Yaskawa INFORM job: X2_34-37(-90,0)_HARDOX.JBI

/JOB
//NAME X2_34-37(-90,0)_HARDOX
//POS
///NPOS 543,543,543,15,0,0
///TOOL 0
///POSTYPE PULSE
///PULSE
C00000=-109615,-71844,-36862,18422,13388,2271
C00001=-107008,40287,15446,7646,74688,11911
C00002=-107149,45804,24218,7788,72161,11701
C00003=-108392,48192,28010,10243,72680,1076
C00004=-108392,48392,29954,10302,71604,983
C00005=-108392,48331,29423,10286,71896,1009
C00006=-108010,50265,31522,10186,71551,1114
C00007=-108392,48331,29423,10286,71896,1009
C00008=-108911,49901,30550,10443,72076,8021
C00009=-109414,51873,32709,10619,71831,7821
C00010=-108911,49901,30550,10443,72076,8021
C00011=-102203,43615,23227,8248,72569,10434
C00012=-106081,49085,29485,15378,74997,2308
C00013=-106081,49206,30588,15419,74401,2232
C00014=-106081,49153,30130,15402,74647,2263
C00015=-105730,50968,32108,15326,74307,2347
C00016=-106081,49153,30130,15402,74647,2263
C00017=-108167,43461,21271,12324,74506,6920
C00018=-107374,42085,15448,7738,75637,11845
C00019=-120191,30165,1303,6226,81332,-6626
C00020=-119709,34887,8992,6124,79003,-6581
C00021=-119523,36874,12198,6088,78043,-6565
C00022=-119519,36825,13807,6108,77033,-6613
C00023=-119523,36874,12198,6088,78043,-6565
C00024=-119515,36764,13496,6103,77191,-6604
C00025=-119868,39633,16467,6214,76866,-6741
C00026=-119515,36764,13496,6103,77191,-6604
C00027=-121889,32841,7793,6759,78864,-7323
C00028=-122776,40716,17165,7052,77228,-7717
C00029=-121823,41691,18182,6780,77023,-7402
C00030=-122776,40716,17165,7052,77228,-7717
C00031=-121889,32783,9008,6775,78090,-7366
C00032=-119523,36874,12198,6088,78043,-6565
C00033=-119709,34887,8992,6124,79003,-6581
C00034=-120191,30165,1303,6226,81332,-6626
C00035=-121604,30205,1144,6630,81559,-7083
C00036=-121089,34887,8794,6520,79231,-7034
C00037=-120696,52216,26132,6337,84983,-6608
C00038=-120696,52210,26931,6339,84491,-6634
C00039=-120890,37827,12979,6483,78156,-7023
C00040=-120878,38017,14560,6499,77285,-7064
C00041=-121214,39658,16269,6601,77105,-7189
C00042=-120878,38555,15116,6500,77220,-7067
C00043=-120100,37082,13567,6272,77355,-6796
C00044=-119528,38122,14634,6107,77190,-6608
C00045=-120486,37092,12834,6373,77838,-6903
C00046=-120682,35058,10322,6419,78351,-6942
C00047=-121186,30266,2562,6523,80690,-6990
C00048=-134026,40869,15057,-4047,52311,-47824
C00049=-133273,45805,23219,-4742,49872,-47398
C00050=-131154,47390,26558,-10411,48349,-46747
C00051=-131420,50658,30105,-10292,47819,-46809
C00052=-130698,69773,43023,-10534,62516,-48132
C00053=-130716,70192,44349,-10580,61922,-48084
C00054=-130716,70230,44981,-10614,61557,-48050
C00055=-130716,70169,43891,-10554,62186,-48109
C00056=-134669,50089,27300,-4593,51640,-48236
C00057=-135826,53842,33106,-2979,47876,-48446
C00058=-135153,55159,34569,-3502,47681,-48138
C00059=-135859,54027,33595,-2932,47595,-48448
C00060=-135721,50610,29531,-3003,48343,-48409
C00061=-134026,40869,15057,-4047,52311,-47824
C00062=-158164,35728,9631,12841,54320,-57618
C00063=-156933,39530,16487,12369,51918,-57402
C00064=-155249,48901,23783,8538,56742,-56466
C00065=-155249,48910,25069,8614,55964,-56530
C00066=-156452,41160,19364,12190,50934,-57317
C00067=-155375,36976,18106,9951,45044,-57856
C00068=-155421,38663,19846,10021,44849,-57900
C00069=-156479,41060,19769,12260,50644,-57365
C00070=-160744,48197,26791,24242,55405,-57248
C00071=-159861,48269,26866,23741,55141,-56924
C00072=-161011,41761,19928,24147,56321,-57142
C00073=-157483,35375,10637,12509,53434,-57446
C00074=-160593,39475,13550,14508,54241,-58615
C00075=-159342,43270,20469,14089,51785,-58436
C00076=-157654,61041,34307,9103,61397,-56807
C00077=-157654,61062,35619,9172,60610,-56871
C00078=-157654,61044,34661,9122,61183,-56824
C00079=-156017,38846,20879,6547,42814,-58158
C00080=-156075,40278,22364,6619,42641,-58197
C00081=-156484,37577,19565,6938,43009,-58369
C00082=-158359,40577,22676,8640,42818,-59307
C00083=-163736,54420,35453,24006,50522,-59362
C00084=-163085,54943,36034,23619,50253,-59126
C00085=-163861,53390,33193,23805,51349,-59211
C00086=-160593,39475,13550,14508,54241,-58615
C00087=-148971,42504,16746,4915,52183,-53021
C00088=-147979,47046,24523,4355,49683,-52716
C00089=-147593,48996,27807,4132,48646,-52593
C00090=-147590,49137,29621,4197,47605,-52637
C00091=-147593,48996,27807,4132,48646,-52593
C00092=-147610,49163,29309,4198,47810,-52637
C00093=-147661,52475,32942,4273,47281,-52683
C00094=-147610,49163,29309,4198,47810,-52637
C00095=-147454,49128,29272,4080,47808,-52567
C00096=-147457,49325,29466,4083,47790,-52569
C00097=-146486,49526,29681,3347,47716,-52137
C00098=-147457,49325,29466,4083,47790,-52569
C00099=-147454,49128,29272,4080,47808,-52567
C00100=-147593,48996,27807,4132,48646,-52593
C00101=-147979,47046,24523,4355,49683,-52716
C00102=-148753,37651,9035,4624,54413,-52827
C00103=-143332,14237,-19618,-15194,67693,-56285
C00104=-143234,13815,-14606,-15619,64520,-55819
C00105=-143234,13420,-12421,-15818,63029,-55609
C00106=-143234,13266,-11275,-15925,62274,-55501
C00107=-143234,13282,-11406,-15913,62359,-55513
C00108=-142905,14636,-10175,-16100,62361,-55388
C00109=-143057,13626,-13166,-15840,63606,-55626
C00110=-122407,-4916,-29077,-25933,68954,-48837
C00111=-79716,14771,-17940,-28940,82202,-34377
C00112=-81521,13206,-15483,-28515,79567,-34389
C00113=-81521,12956,-14255,-28586,78787,-34193
C00114=-81536,13061,-14375,-28568,78899,-34239
C00115=-81552,13376,-14091,-28564,78881,-34239
C00116=-81324,12822,-15528,-28589,79487,-34301
C00117=-153828,-54456,-66092,3136,64230,-58148
C00118=-168903,-101217,-87597,11823,54897,-64642
C00119=-187075,-120078,-80481,24912,5471,-74731
C00120=-125084,-120078,-92282,24912,5045,-74731
C00121=-122155,56416,27906,-88,21317,-63492
C00122=-122155,75596,27906,-2527,72055,-63492
C00123=-129231,63588,14742,9851,74193,-63747
C00124=-129934,64141,19195,10317,71853,-64173
C00125=-129934,63674,20017,10359,71118,-64236
C00126=-129934,63737,19901,10353,71221,-64227
C00127=-129659,64892,21241,10232,70961,-64158
C00128=-129934,64415,18756,10296,72257,-64138
C00129=-132222,69706,24963,11475,71461,-64978
C00130=-132222,69058,26180,11545,70402,-65080
C00131=-131900,68421,25429,11378,70491,-64961
C00132=-131996,66718,21836,11340,71814,-64867
C00133=-130068,63875,18521,10367,72141,-64191
C00134=-129934,63737,19901,10353,71221,-64227
C00135=-129659,64892,21241,10232,70961,-64158
C00136=-129936,63793,17790,10283,72529,-64117
C00137=-88784,58262,10938,-10282,73900,-50815
C00138=-84208,56991,12900,-3171,67181,-46725
C00139=-84435,57608,15935,-3079,65626,-46760
C00140=-84435,57210,16828,-3097,64873,-46739
C00141=-84435,57270,16685,-3094,64991,-46743
C00142=-84516,58633,18225,-3054,64742,-46763
C00143=-84215,57626,14285,-3179,66658,-46710
C00144=-88784,58262,10938,-10282,73900,-50815
C00145=-130230,57807,7300,10270,75892,-63928
C00146=-119131,59701,11284,-18823,72688,-66064
C00147=-121021,64874,21663,-18257,68751,-66091
C00148=-121021,64408,22622,-18356,67963,-65965
C00149=-121021,64908,21591,-18251,68811,-66098
C00150=-119131,67163,24223,-19268,68781,-65421
C00151=-119066,66124,24431,-19384,68169,-65294
C00152=-119315,66407,24761,-19266,68060,-65365
C00153=-119315,66969,23588,-19142,69017,-65526
C00154=-121021,64979,21457,-18238,68923,-66116
C00155=-121021,64479,22465,-18340,68089,-65984
C00156=-120883,66044,24287,-18448,67818,-65890
C00157=-120883,66039,23301,-18376,68392,-65982
C00158=-125359,68164,24258,-15996,67985,-67508
C00159=-125355,67935,25342,-16085,67231,-67400
C00160=-125355,67510,26289,-16176,66462,-67291
C00161=-125355,67568,26150,-16162,66575,-67307
C00162=-125232,69006,27841,-16263,66308,-67224
C00163=-125264,67856,24082,-16054,67958,-67468
C00164=-118603,65727,21589,-19430,69736,-65391
C00165=-117191,86264,44946,-23194,75505,-66935
C00166=-117189,86115,44761,-23192,75540,-66941
C00167=-117189,86115,44761,-23192,75540,-66941
C00168=-117506,84477,42726,-23036,75832,-67112
C00169=-117132,73456,32688,-25561,71261,-66383
C00170=-118175,73897,33217,-25111,70866,-66682
C00171=-123739,77574,37647,-22686,68558,-68266
C00172=-123019,74931,32102,-22743,70649,-68420
C00173=-118383,77560,28081,-24424,75407,-67742
C00174=-128287,78191,30299,3222,75938,-66053
C00175=-128503,77276,32915,3346,73869,-66179
C00176=-128483,76731,32333,3336,73949,-66169
C00177=-128483,76731,32333,3336,73949,-66169
C00178=-128335,75085,30341,3266,74321,-66111
C00179=-127967,73943,28963,3095,74566,-65984
C00180=-126238,72254,26940,2321,74892,-65413
C00181=-107561,64945,18412,-6002,76780,-59423
C00182=-95850,66897,26093,8333,67040,-51862
C00183=-95804,66521,24248,8255,67969,-51781
C00184=-109126,32483,-12900,14644,74981,-55562
C00185=-109126,32483,-12900,14644,28895,-55562
C00186=-105965,-15733,-41727,12755,21555,-55066
C00187=-95466,-93835,-85705,-21780,8598,-39995
C00188=-117456,-93835,-85705,-3320,8456,-83429
C00189=-140967,-12970,-52901,4588,62048,-69725
C00190=-151426,22553,-30287,8605,79970,-63791
C00191=-170197,65047,13937,16074,97750,-54995
C00192=-169007,70240,20067,15770,96475,-54777
C00193=-175404,86334,34832,19373,106938,-55773
C00194=-174173,83341,34513,19133,105400,-55601
C00195=-179433,56900,11422,30057,94253,-55502
C00196=-178535,49502,4014,27996,88823,-56876
C00197=-179527,69319,26237,30671,91177,-56324
C00198=-179117,69620,25739,29739,90864,-56355
C00199=-180097,67994,26330,32410,86483,-57198
C00200=-174100,64042,14056,17976,91926,-56289
C00201=-175447,65123,11808,18399,94042,-56406
C00202=-164161,72,-39985,-6764,90046,-34295
C00203=-130432,-55243,-47386,-13424,82603,8412
C00204=-110572,-56965,-55890,-14658,90278,14468
C00205=-134387,-39172,-38807,12376,86277,-20344
C00206=-136266,-41846,-34601,16059,78566,-27361
C00207=-135424,-39022,-31748,15965,78109,-27121
C00208=-132144,-43884,-34748,15569,76844,-26110
C00209=-133349,-52476,-37829,19150,70304,-22714
C00210=-132707,-53219,-38228,19044,70026,-22517
C00211=-133874,-49344,-36092,21066,73724,-26553
C00212=-127403,-56601,-39797,20204,70737,-24655
C00213=-130575,-58808,-42172,20683,71834,-25657
C00214=-131419,-52897,-41760,13173,72105,-2236
C00215=-151757,-37235,-32664,25855,92713,-16023
C00216=-148694,-31120,-30848,28555,97484,-16481
C00217=-152363,20888,-11521,23566,108052,-25705
C00218=-155491,63274,13853,18429,111086,-34801
C00219=-150514,89045,46229,21307,107758,-32982
C00220=-149106,88504,48693,21100,105732,-32842
C00221=-152517,63826,23946,30540,100235,-10367
C00222=-144965,57793,12440,13988,97767,-10863
C00223=-145698,58452,15092,12206,89625,-12161
C00224=-143897,56959,13401,8510,88242,-7863
C00225=-138738,54288,10428,-948,87223,2685
C00226=-138154,54736,10996,-4550,87493,6522
C00227=-140559,38499,-1659,880,75847,28463
C00228=-140619,46287,2526,1728,82676,28626
C00229=-139837,43342,-3801,1439,85041,28899
C00230=-141798,27002,-27786,2149,91441,28405
C00231=-143772,-19107,-38740,14355,94017,-12677
C00232=-143698,-35148,-33847,20276,92427,-33189
C00233=-141918,-24797,-26817,20326,92921,-32464
C00234=-139594,-23350,-22642,20301,90627,-32011
C00235=-137429,-46971,-35033,19650,72370,-30958
C00236=-130857,-51491,-37639,10003,64087,-16893
C00237=-124996,-53139,-38566,2264,61948,-7877
C00238=-114020,-50430,-37038,-13344,65966,10499
C00239=-112071,-46775,-34852,-17581,69897,16673
C00240=-117935,-60108,-42034,-7672,56240,37337
C00241=-115664,-65010,-47736,-8512,57449,38158
C00242=-121785,-61828,-52329,-5505,69210,35118
C00243=-148930,-33628,-41038,4538,77484,18447
C00244=-163858,24222,1645,10794,81228,7547
C00245=-163712,28964,9442,10824,78886,7392
C00246=-163731,31317,12909,10857,77980,7305
C00247=-164778,31926,13518,11115,78061,6949
C00248=-169796,40183,22289,16135,80950,-18095
C00249=-170946,41436,24303,16621,77711,-36979
C00250=-169129,60932,43860,12206,77205,-36613
C00251=-174700,53660,39403,25265,70725,-61619
C00252=-176244,52382,34806,25393,73168,-61673
C00253=-174832,57379,31343,14926,87681,-59388
C00254=-147451,1111,-29714,5377,100632,-19781
C00255=-112791,-31989,-50015,-2241,90212,24459
C00256=-107981,-35875,-46971,-4517,78040,26268
C00257=-109410,-31915,-41181,-4141,76439,25836
C00258=-109671,-29943,-38250,-4081,75635,25773
C00259=-108634,-25346,-36028,-8315,81190,19632
C00260=-113738,-28838,-38579,-3049,79626,8435
C00261=-120146,-28716,-38356,4151,79685,-1679
C00262=-130395,-15154,-28625,15552,87688,-20481
C00263=-128753,-14804,-28536,10287,83416,-20949
C00264=-132110,-20936,-30028,13610,74111,-31363
C00265=-127631,-24253,-35023,5775,74490,-30240
C00266=-129181,-27934,-40726,6212,76213,-30690
C00267=-139651,-3107,-33687,4364,86662,15844
C00268=-140099,618,-27389,4493,84729,15631
C00269=-139376,8672,-20712,3285,88556,15837
C00270=-139238,10495,-19621,-120,90504,9397
C00271=-144296,12055,-18225,6153,91589,-773
C00272=-148325,17435,-13208,10971,94126,-9741
C00273=-150411,23892,-7112,13293,96134,-15177
C00274=-151318,31111,-42,13381,95653,-15535
C00275=-151917,36538,5447,13433,95174,-15789
C00276=-152712,20066,-9195,12847,84122,-38020
C00277=-154297,18366,-13942,13242,86364,-38311
C00278=-149036,10060,-28234,-4051,95048,45397
C00279=-110442,-7238,-41801,-11532,98024,57505
C00280=-109513,-32833,-49968,-8912,71006,60642
C00281=-108272,-31490,-45832,-9532,69313,61212
C00282=-121999,-28446,-43764,-3614,68504,56397
C00283=-145834,-8654,-29251,6781,70208,48084
C00284=-161078,10619,-11723,7061,67590,41743
C00285=-161402,9669,-16363,7100,69967,41771
C00286=-143466,6998,19042,5158,32162,-41222
C00287=-147237,-51968,-50099,-4175,73083,-42408
C00288=3643,-76224,-106676,19950,71810,76872
C00289=6047,-95755,-92046,-14751,98253,9605
C00290=8024,-164446,-133802,-16041,6272,12396
C00291=8024,-164446,-133802,-16041,6272,12396
C00292=80911,-131071,-112390,-19160,57527,-4768
C00293=107387,-112645,-89313,-18613,48039,-3448
C00294=120529,-94925,-67119,-18087,38914,-2179
C00295=102807,-11704,-32462,-5874,76695,-13415
C00296=103436,-3791,-23255,-6127,75148,-13126
C00297=103560,-1765,-20423,-6188,74460,-13051
C00298=103560,-1806,-19122,-6212,73642,-13010
C00299=103601,-1431,-19452,-6214,74041,-13015
C00300=104452,277,-18031,-6506,74110,-12725
C00301=103539,-2063,-20212,-6189,74177,-13043
C00302=120126,-10436,-31938,-6011,80471,6680
C00303=119034,-8056,-29018,-5697,79822,6345
C00304=119034,-8150,-28117,-5707,79221,6375
C00305=119034,-8056,-29018,-5697,79822,6345
C00306=118636,-7203,-28340,-5579,79816,6211
C00307=119064,-5644,-27091,-5704,79877,6351
C00308=118636,-7203,-28340,-5579,79816,6211
C00309=122253,-9472,-30321,-6643,80135,7408
C00310=122707,-2954,-24944,-6773,80213,7552
C00311=122021,-2022,-23613,-6578,79819,7343
C00312=122707,-3013,-24427,-6779,79866,7571
C00313=121204,9301,-16198,-6319,81003,7011
C00314=120827,28505,-838,-6150,90516,6420
C00315=120827,28295,458,-6147,89615,6464
C00316=120979,11415,-12534,-6272,79823,6996
C00317=121673,13624,-10544,-6477,79786,7230
C00318=120979,11542,-13540,-6262,80500,6963
C00319=121039,12182,-11846,-8037,80321,9006
C00320=120294,13253,-10880,-7825,80206,8763
C00321=121039,12182,-11846,-8037,80321,9006
C00322=121310,5674,-20943,-6336,82061,6993
C00323=139815,-25323,-43479,-19,53677,50237
C00324=135350,7914,-23933,5265,75592,49702
C00325=135350,7716,-23321,5277,75113,49682
C00326=137572,-18164,-33682,1617,51348,49297
C00327=138000,-16627,-32540,1306,51428,49477
C00328=137572,-18164,-33682,1617,51348,49297
C00329=141541,-18151,-35068,-1262,52202,50952
C00330=141186,-12326,-28968,-1018,51433,50811
C00331=140737,-11536,-28358,-690,51458,50623
C00332=141186,-12326,-28968,-1018,51433,50811
C00333=159686,26179,2441,-14066,53601,58348
C00334=155838,47235,15677,-4337,69179,56490
C00335=155838,47134,16315,-4350,68734,56506
C00336=159232,27229,5186,-13963,52408,58323
C00337=159232,27225,5485,-13997,52227,58349
C00338=159220,29212,7438,-14024,52052,58369
C00339=159232,27225,5485,-13997,52227,58349
C00340=164735,35698,13654,-29808,58437,68077
C00341=164028,35618,13572,-29436,58200,67836
C00342=164735,35698,13654,-29808,58437,68077
C00343=157023,57493,24423,-2651,73609,57035
C00344=157023,57387,25075,-2656,73154,57045
C00345=161795,29787,7764,-15728,52595,59373
C00346=161783,31729,9695,-15761,52409,59396
C00347=161795,29787,7764,-15728,52595,59373
C00348=163888,29194,5832,-16938,53858,60057
C00349=165806,38731,16984,-22046,53706,63214
C00350=165192,38605,16853,-21659,53559,62976
C00351=165806,38731,16984,-22046,53706,63214
C00352=161708,46386,23154,-8907,61269,44547
C00353=161224,48066,26131,-8737,60259,44442
C00354=161222,48202,27939,-8826,59228,44523
C00355=161224,48066,26131,-8737,60259,44442
C00356=161238,48238,27638,-8816,59431,44513
C00357=161118,51495,31180,-8798,58918,44508
C00358=161238,48238,27638,-8816,59431,44513
C00359=161086,48113,27502,-8735,59433,44454
C00360=161078,48307,27691,-8732,59416,44452
C00361=160108,47930,27281,-8216,59373,44078
C00362=161078,48307,27691,-8732,59416,44452
C00363=161086,48113,27502,-8735,59433,44454
C00364=161224,48066,26131,-8737,60259,44442
C00365=161708,46386,23154,-8907,61269,44547
C00366=162944,42495,16096,-9351,63722,44812
C00367=163630,17067,-13667,4112,73791,46186
C00368=159524,23907,-3320,12553,74764,46006
C00369=159524,23795,-2481,12584,74204,45948
C00370=159524,23816,-2646,12579,74314,45960
C00371=159245,24593,-1899,12687,74295,45862
C00372=159194,24027,-3919,12653,75231,45943
C00373=111493,-14143,-36721,26833,87177,31237
C00374=87125,287,-27276,31139,96728,24609
C00375=86989,1093,-24681,31070,95757,24290
C00376=87014,942,-23026,30995,94803,24037
C00377=87014,978,-23253,31006,94939,24075
C00378=87144,2304,-22132,30991,94887,24109
C00379=86824,1101,-25587,31137,96301,24374
C00380=101451,-10960,-35317,28856,91089,28489
C00381=120471,-127745,-104072,26282,69111,30519
C00382=120473,-120954,-92945,26872,66091,29789
C00383=120482,-116919,-91462,23600,9236,-68753
C00384=120620,4301,-23209,7431,28987,-61255
C00385=120635,53932,-6539,3654,81089,-58599
C00386=136219,23700,-29963,-4017,80003,-54068
C00387=137871,24187,-22740,-4910,75904,-53421
C00388=137871,23434,-21830,-4928,74961,-53382
C00389=137871,24024,-22549,-4915,75706,-53414
C00390=134128,22508,-24006,-3048,75657,-54576
C00391=134008,21904,-23397,-2994,74967,-54596
C00392=135424,22939,-22404,-3704,74941,-54154
C00393=135424,23559,-23154,-3692,75720,-54178
C00394=137871,24102,-22640,-4913,75801,-53417
C00395=137871,23511,-21927,-4928,75061,-53388
C00396=137660,24371,-21096,-4823,74982,-53451
C00397=137740,24894,-23570,-4829,76771,-53495
C00398=141619,27919,-20548,-6751,76714,-52296
C00399=141520,27933,-18669,-6730,75567,-52267
C00400=141520,27387,-17987,-6751,74870,-52228
C00401=141520,27457,-18077,-6749,74961,-52234
C00402=141319,28424,-17122,-6652,74858,-52293
C00403=141474,28149,-19863,-6687,76406,-52330
C00404=142787,22165,-27593,-22317,81169,-54825
C00405=128980,17445,-27826,5941,73245,-72607
C00406=128980,16959,-27218,5961,72624,-72637
C00407=128980,17663,-28087,5933,73516,-72592
C00408=131920,22243,-23763,4387,73040,-71685
C00409=131830,21695,-23039,4452,72319,-71739
C00410=131353,21345,-23370,4704,72369,-71890
C00411=131353,21989,-24168,4684,73188,-71859
C00412=128980,17788,-28233,5930,73669,-72585
C00413=128980,17036,-27317,5957,72724,-72631
C00414=128670,17969,-26451,6125,72689,-72731
C00415=128750,17329,-29580,6037,74272,-72626
C00416=130234,20174,-32481,-12163,78976,-77377
C00417=120812,3159,-42178,-18150,73789,-82874
C00418=118792,1921,-39571,-17276,71261,-83158
C00419=118792,1177,-38518,-17376,70275,-83012
C00420=118792,1261,-38644,-17364,70392,-83030
C00421=118719,2466,-37625,-17328,70371,-83052
C00422=118706,2074,-39642,-17220,71363,-83204
C00423=136219,23700,-29963,-4017,80003,-54068
C00424=135146,53480,-2149,-5253,96368,-48776
C00425=135068,55927,1059,-5224,95649,-48768
C00426=135523,55672,2883,-5335,94427,-48578
C00427=135661,54651,1734,-5376,94618,-48548
C00428=135661,54651,1734,-5376,94618,-48548
C00429=135983,53920,911,-5466,94767,-48457
C00430=136620,53721,687,-5642,94843,-48267
C00431=137961,48169,-4011,-6751,91428,-47860
C00432=136603,56271,5440,5574,93005,-31091
C00433=135971,53463,1330,5761,94127,-31234
C00434=136155,41032,-15285,-5561,98105,-48550
C00435=137845,50680,-6420,-9428,103493,20009
C00436=141337,57917,4429,-10007,100945,21296
C00437=140502,58531,6185,-9812,100106,21104
C00438=140613,57301,4783,-9843,100345,21119
C00439=140627,56270,3706,-9850,100477,21113
C00440=140579,56145,3582,-9841,100484,21097
C00441=140334,55501,2947,-9795,100521,21013
C00442=138250,53530,591,-9675,101364,17502
C00443=117794,38005,-16358,-5505,102094,11159
C00444=108286,34694,-16144,-16728,96590,5594
C00445=108161,32376,-20470,-16766,97976,5364
C00446=125216,14187,-38215,-21178,102884,9957
C00447=125216,14187,-17583,-21178,28179,9957
C00448=133106,-138478,-90488,-65593,16001,37631
C00449=133106,-138478,-90488,-65593,-54320,37631
C00450=133106,-138478,-104097,-150628,-10334,-7073
C00451=133106,-138478,-104097,-1528,-10334,-7073
C00452=146394,-11991,-35742,-1101,69372,37360
C00453=151186,4741,-23090,-4031,73296,40716
C00454=156388,23931,-10315,-7169,81629,44228
C00455=174995,75619,44100,-18565,95741,57403
C00456=178295,72858,49572,-29598,87914,53870
C00457=178363,71681,49458,-30316,81279,55416
C00458=178775,74747,53745,-31442,79609,55982
C00459=178120,80280,53499,-25679,87195,54196
C00460=177788,66292,45128,-22799,80541,57078
C00461=165876,20944,-7359,-14016,91072,47752
C00462=144031,-8096,-47002,481,102749,33013
C00463=113249,-55125,-55779,6617,87879,-14622
C00464=105402,-49476,-43093,17129,78821,-17705
C00465=107372,-45114,-37354,16923,77172,-17229
C00466=107897,-43226,-34630,16890,76385,-17150
C00467=123036,-54169,-41018,-3647,66196,-9526
C00468=125103,-54109,-40569,-7539,65613,-9158
C00469=133018,-52183,-38196,-18552,67287,-3963
C00470=135096,-56008,-41994,-19101,68310,-3149
C00471=148619,-36280,-33179,-26254,90102,11601
C00472=132022,-46525,-51369,-8915,93592,12104
C00473=152394,4325,-31091,-21424,100011,27739
C00474=150620,74441,30669,-21497,109248,32750
C00475=152126,53384,9711,-25318,101313,34092
C00476=150816,58410,15272,-25509,99566,10610
C00477=152757,73148,32936,-27341,97295,8053
C00478=150720,57278,15123,-23866,91102,-1332
C00479=147911,49489,6323,-18230,87408,-8983
C00480=145167,44213,390,-9981,84631,-17850
C00481=142774,42237,-1321,-4504,82417,-25550
C00482=141310,41249,-3509,-1904,83312,-28397
C00483=140520,38377,-9680,-1608,85617,-28672
C00484=145482,-30493,-50756,-14636,95383,13188
C00485=142176,-26033,-28146,-20229,92686,32606
C00486=139838,-24569,-23969,-20194,90398,32145
C00487=141333,-43488,-32424,-24355,75177,35516
C00488=142946,-39788,-29545,-27566,77515,12382
C00489=142712,-38988,-29426,-26650,76094,9122
C00490=137490,-51139,-36024,-22440,64589,-1384
C00491=129219,-61272,-40095,-12800,52551,-14455
C00492=125098,-62268,-41395,-3949,52110,-22670
C00493=120434,-59895,-41306,5152,54802,-34175
C00494=118218,-60267,-42467,7826,55944,-37248
C00495=115940,-65207,-48159,8687,57132,-38075
C00496=158051,-33814,-49892,-7441,80913,-13725
C00497=163513,25616,3177,-10792,80459,-7597
C00498=163372,30455,11081,-10830,78103,-7439
C00499=163993,28142,11085,-12803,74423,-6981
C00500=161648,29238,11147,-4496,75447,-179
C00501=171143,45412,28292,-19077,81279,23270
C00502=173705,65046,50293,-22854,85176,36170
C00503=173974,62485,49606,-24076,73199,49227
C00504=172570,70781,55370,-19160,78152,47867
C00505=174025,68948,50025,-19270,80716,47984
C00506=170072,38309,9009,-5458,81396,48416
C00507=145937,-33300,-50613,-2555,87892,10434
C00508=117969,-26674,-50251,1455,96093,-22658
C00509=108065,-36096,-47601,4778,77881,-26213
C00510=109507,-32110,-41823,4391,76297,-25779
C00511=109013,-37865,-42571,5415,69231,-26193
C00512=107679,-33877,-40967,9851,74714,-20356
C00513=113110,-32097,-41032,3661,77261,-8676
C00514=119719,-29513,-40298,-3828,79988,1546
C00515=130402,-22376,-34110,-15555,82843,20591
C00516=132503,-6978,-23545,-15597,88653,21115
C00517=133170,-4219,-21374,-15691,88857,21320
C00518=127848,-25408,-36231,-5685,74178,30350
C00519=129407,-29126,-41925,-6135,75876,30806
C00520=139811,-3516,-34603,-4319,86523,-15767
C00521=140259,233,-28314,-4452,84609,-15556
C00522=139695,2013,-26001,-4296,84073,-15716
C00523=138357,5138,-24127,1260,87157,-9766
C00524=142581,5877,-23634,-3711,87883,1101
C00525=150814,13398,-16280,-14778,91025,16227
C00526=153586,30573,-617,-18226,97890,27109
C00527=154794,42487,11468,-18272,96901,27676
C00528=154809,42525,11398,-18275,96963,27672
C00529=153093,18834,-10833,-12947,84050,38162
C00530=154693,17143,-15552,-13354,86281,38457
C00531=130444,-10965,-45057,12181,91290,25722
C00532=107975,-11927,-39534,17315,91376,18359
C00533=106451,-5636,-31397,17601,89993,17646
C00534=108649,-4402,-29158,22134,89122,18947
C00535=144880,18547,-8956,13065,80859,30158
C00536=145078,17418,-12459,12964,82365,30383
C00537=149017,-29902,-48296,-21465,64483,30019
C00538=102406,-109115,-77602,-2898,35707,-11807
C00539=80911,-131071,-112390,-19160,57527,-4768
C00540=8024,-164446,-133802,-16041,6272,12396
C00541=8024,-164446,-133802,-16041,6272,12396
C00542=1579,-114561,-88072,141,60969,-160
BC00000=287767,672594,392898
BC00001=287767,702390,199743
BC00002=287767,702390,199743
BC00003=287767,702390,199743
BC00004=287767,702390,199743
BC00005=287767,702390,199743
BC00006=287767,702390,199743
BC00007=287767,702390,199743
BC00008=287767,702390,199743
BC00009=287767,702390,199743
BC00010=287767,702390,199743
BC00011=287767,702390,199743
BC00012=287767,702390,199743
BC00013=287767,702390,199743
BC00014=287767,702390,199743
BC00015=287767,702390,199743
BC00016=287767,702390,199743
BC00017=287767,702390,199743
BC00018=287767,702390,199743
BC00019=325466,709124,183073
BC00020=325466,709124,183073
BC00021=325466,709124,183073
BC00022=325466,709124,183073
BC00023=325466,709124,183073
BC00024=325466,709124,183073
BC00025=325466,709124,183073
BC00026=325466,709124,183073
BC00027=325466,709124,183073
BC00028=325466,709124,183073
BC00029=325466,709124,183073
BC00030=325466,709124,183073
BC00031=325466,709124,183073
BC00032=325466,709124,183073
BC00033=325466,709124,183073
BC00034=325466,709124,183073
BC00035=304409,729721,181352
BC00036=304409,729721,181352
BC00037=304409,729721,181352
BC00038=304409,729721,181352
BC00039=304409,729721,181352
BC00040=304409,729721,181352
BC00041=304409,729721,181352
BC00042=304409,729721,181352
BC00043=304409,729721,181352
BC00044=304409,729721,181352
BC00045=304409,729721,181352
BC00046=304409,729721,181352
BC00047=304409,729721,181352
BC00048=360941,686135,119054
BC00049=360941,686135,119054
BC00050=360941,686135,119054
BC00051=360941,686135,119054
BC00052=360941,686135,119054
BC00053=360941,686135,119054
BC00054=360941,686135,119054
BC00055=360941,686135,119054
BC00056=360941,686135,119054
BC00057=360941,686135,119054
BC00058=360941,686135,119054
BC00059=360941,686135,119054
BC00060=360941,686135,119054
BC00061=360941,686135,119054
BC00062=398174,742009,118025
BC00063=398174,742009,118025
BC00064=398174,742009,118025
BC00065=398174,742009,118025
BC00066=398174,742009,118025
BC00067=398174,742009,118025
BC00068=398174,742009,118025
BC00069=398174,742009,118025
BC00070=398174,742009,118025
BC00071=398174,742009,118025
BC00072=398174,742009,118025
BC00073=398174,742009,118025
BC00074=397434,738268,118311
BC00075=397434,738268,118311
BC00076=397434,738268,118311
BC00077=397434,738268,118311
BC00078=397434,738268,118311
BC00079=397434,738268,118311
BC00080=397434,738268,118311
BC00081=397434,738268,118311
BC00082=397434,738268,118311
BC00083=397434,738268,118311
BC00084=397434,738268,118311
BC00085=397434,738268,118311
BC00086=397434,738268,118311
BC00087=337757,747913,121043
BC00088=337757,747913,121043
BC00089=337757,747913,121043
BC00090=337757,747913,121043
BC00091=337757,747913,121043
BC00092=337757,747913,121043
BC00093=337757,747913,121043
BC00094=337757,747913,121043
BC00095=337757,747913,121043
BC00096=337757,747913,121043
BC00097=337757,747913,121043
BC00098=337757,747913,121043
BC00099=337757,747913,121043
BC00100=337757,747913,121043
BC00101=337757,747913,121043
BC00102=337757,747913,121043
BC00103=337757,747913,121043
BC00104=337757,747913,121043
BC00105=337757,747913,121043
BC00106=337757,747913,121043
BC00107=337757,747913,121043
BC00108=337757,747913,121043
BC00109=337757,747913,121043
BC00110=337757,747913,121043
BC00111=235567,747913,121043
BC00112=235567,747913,121043
BC00113=235567,747913,121043
BC00114=235567,747913,121043
BC00115=235567,747913,121043
BC00116=235567,747913,121043
BC00117=345966,747913,121043
BC00118=345966,747913,121043
BC00119=345966,747913,121043
BC00120=143697,705044,13
BC00121=143697,705044,13
BC00122=143697,705044,13
BC00123=143697,705044,13
BC00124=143697,705044,13
BC00125=143697,705044,13
BC00126=143697,705044,13
BC00127=143697,705044,13
BC00128=143697,705044,13
BC00129=143697,705044,13
BC00130=143697,705044,13
BC00131=143697,705044,13
BC00132=143697,705044,13
BC00133=143697,705044,13
BC00134=143697,705044,13
BC00135=143697,705044,13
BC00136=143697,705044,13
BC00137=65691,720245,4426
BC00138=65691,720245,4426
BC00139=65691,720245,4426
BC00140=65691,720245,4426
BC00141=65691,720245,4426
BC00142=65691,720245,4426
BC00143=65691,720245,4426
BC00144=65691,720245,4426
BC00145=143697,705044,13
BC00146=143697,705044,13
BC00147=143697,705044,13
BC00148=143697,705044,13
BC00149=143697,705044,13
BC00150=143697,705044,13
BC00151=143697,705044,13
BC00152=143697,705044,13
BC00153=143697,705044,13
BC00154=143697,705044,13
BC00155=143697,705044,13
BC00156=143697,705044,13
BC00157=143697,705044,13
BC00158=143697,705044,13
BC00159=143697,705044,13
BC00160=143697,705044,13
BC00161=143697,705044,13
BC00162=143697,705044,13
BC00163=143697,705044,13
BC00164=143697,705044,13
BC00165=143697,705044,13
BC00166=143697,705044,13
BC00167=143697,705044,13
BC00168=143697,705044,13
BC00169=143697,705044,13
BC00170=143697,705044,13
BC00171=143697,705044,13
BC00172=143697,705044,13
BC00173=143697,705044,13
BC00174=143697,705044,13
BC00175=143697,705044,13
BC00176=143697,705044,13
BC00177=143697,705044,13
BC00178=143697,705044,13
BC00179=143697,705044,13
BC00180=143697,705044,13
BC00181=143697,705044,13
BC00182=99716,705044,13
BC00183=99716,705044,13
BC00184=99716,705044,13
BC00185=99716,705044,13
BC00186=99716,705044,13
BC00187=99716,663642,13
BC00188=314973,663642,13
BC00189=345769,722785,14347
BC00190=359469,749095,20724
BC00191=382499,793323,31443
BC00192=382499,793323,31443
BC00193=398174,809232,53
BC00194=398174,809232,53
BC00195=398174,809232,53
BC00196=398174,809232,53
BC00197=398174,809232,53
BC00198=398174,809232,53
BC00199=398174,809232,53
BC00200=398174,809232,53
BC00201=398174,809232,53
BC00202=378399,812249,125880
BC00203=350148,816882,305631
BC00204=350148,816882,305631
BC00205=350717,816957,305463
BC00206=350717,816957,305463
BC00207=350717,816957,305463
BC00208=350717,816957,305463
BC00209=350717,816957,305459
BC00210=350717,816957,305459
BC00211=350717,816957,305459
BC00212=350717,816957,305459
BC00213=350717,816957,305459
BC00214=350717,816957,305463
BC00215=350717,816957,305463
BC00216=350148,816882,305631
BC00217=357486,783574,171223
BC00218=363745,755164,56581
BC00219=350108,749289,42117
BC00220=350108,749289,42117
BC00221=350108,749289,42114
BC00222=350108,749289,42117
BC00223=350108,749289,42117
BC00224=350108,749289,42117
BC00225=350108,749289,42117
BC00226=350108,749289,42117
BC00227=350108,749289,42117
BC00228=350108,749289,42117
BC00229=350108,749289,42117
BC00230=350045,748919,44151
BC00231=332829,802151,218589
BC00232=324221,828766,305808
BC00233=324283,829135,303773
BC00234=324283,829135,303773
BC00235=324283,829135,303773
BC00236=324283,829135,303773
BC00237=324283,829135,303773
BC00238=324283,829135,303773
BC00239=324283,829135,303773
BC00240=324283,829135,303773
BC00241=324283,829135,303773
BC00242=324221,828766,305808
BC00243=365904,809152,256676
BC00244=398174,795215,220015
BC00245=398174,795215,220015
BC00246=398174,795215,220015
BC00247=398174,795215,220015
BC00248=398174,795215,220015
BC00249=398174,795215,220015
BC00250=398174,795215,220015
BC00251=398174,795215,220015
BC00252=398174,795215,220015
BC00253=398174,795215,220015
BC00254=365121,791381,219974
BC00255=328869,787176,219929
BC00256=328869,787176,219929
BC00257=328869,787176,219929
BC00258=328869,787176,219929
BC00259=328869,787176,219929
BC00260=328869,787176,219929
BC00261=328869,787176,219929
BC00262=328869,787176,219929
BC00263=328869,787176,219929
BC00264=328869,787176,219929
BC00265=328869,787176,219929
BC00266=328869,787176,219929
BC00267=366743,775181,149862
BC00268=366743,775181,149862
BC00269=366743,775181,149862
BC00270=366743,775181,149862
BC00271=366743,775181,149862
BC00272=366743,775181,149862
BC00273=366743,775181,149862
BC00274=366743,775181,149862
BC00275=366743,775181,149862
BC00276=366743,775181,149862
BC00277=366743,775181,149862
BC00278=366743,775181,149862
BC00279=319910,775181,156236
BC00280=319910,775181,156236
BC00281=319910,775181,156236
BC00282=319910,775181,156236
BC00283=319910,775181,156236
BC00284=361358,775181,156236
BC00285=361358,775181,156236
BC00286=366743,675039,355777
BC00287=366743,675039,355777
BC00288=199464,674570,1075173
BC00289=95044,675039,919146
BC00290=95044,675039,1075229
BC00291=235813,1345575,1075229
BC00292=291733,1363613,501241
BC00293=295042,1365829,344881
BC00294=288108,1367960,194507
BC00295=288108,1365832,194507
BC00296=288108,1369193,194507
BC00297=288108,1369264,194507
BC00298=288108,1369264,194507
BC00299=288108,1369614,194507
BC00300=288108,1369614,194507
BC00301=288108,1368913,194507
BC00302=325834,1368698,177132
BC00303=325834,1367902,177132
BC00304=325834,1367902,177132
BC00305=325834,1367902,177132
BC00306=325834,1367902,177132
BC00307=325834,1367902,177132
BC00308=325834,1367902,177132
BC00309=325834,1368223,177132
BC00310=325834,1368768,177132
BC00311=325834,1368768,177132
BC00312=325834,1368768,177132
BC00313=304798,1367887,175873
BC00314=304798,1368278,175873
BC00315=304798,1368278,175873
BC00316=304798,1368278,175873
BC00317=304798,1368278,175873
BC00318=304798,1368278,175873
BC00319=304798,1368278,175873
BC00320=304798,1368278,175873
BC00321=304798,1368278,175873
BC00322=304798,1368714,175873
BC00323=360316,1368040,111260
BC00324=360316,1367747,111260
BC00325=360316,1367747,111260
BC00326=360316,1367747,111260
BC00327=360316,1367747,111260
BC00328=360316,1367747,111260
BC00329=360316,1368265,111260
BC00330=360316,1367537,111260
BC00331=360316,1367537,111260
BC00332=360316,1367537,111260
BC00333=398174,1367762,110837
BC00334=398174,1365917,110837
BC00335=398174,1365917,110837
BC00336=398174,1365917,110837
BC00337=398174,1365917,110837
BC00338=398174,1365917,110837
BC00339=398174,1365917,110837
BC00340=398174,1365917,110837
BC00341=398174,1365917,110837
BC00342=398174,1365917,110837
BC00343=397184,1368437,111272
BC00344=397184,1368437,111272
BC00345=397184,1368437,111272
BC00346=397184,1368437,111272
BC00347=397184,1368437,111272
BC00348=397184,1367234,111272
BC00349=397184,1367282,111272
BC00350=397184,1367282,111272
BC00351=397184,1367282,111272
BC00352=375501,1345864,156348
BC00353=375501,1345864,156348
BC00354=375501,1345864,156348
BC00355=375501,1345864,156348
BC00356=375501,1345864,156348
BC00357=375501,1345864,156348
BC00358=375501,1345864,156348
BC00359=375501,1345864,156348
BC00360=375501,1345864,156348
BC00361=375501,1345864,156348
BC00362=375501,1345864,156348
BC00363=375501,1345864,156348
BC00364=375501,1345864,156348
BC00365=375501,1345864,156348
BC00366=375501,1345864,156348
BC00367=375501,1345864,156348
BC00368=375501,1345864,156348
BC00369=375501,1345864,156348
BC00370=375501,1345864,156348
BC00371=375501,1345864,156348
BC00372=375501,1345864,156348
BC00373=299838,1345863,156346
BC00374=273619,1345863,156346
BC00375=273619,1345863,156346
BC00376=273619,1345863,156346
BC00377=273619,1345863,156346
BC00378=273619,1345863,156346
BC00379=273619,1345863,156346
BC00380=273619,1345863,156346
BC00381=319522,1369258,95050
BC00382=171115,1369889,1882
BC00383=171115,1369889,1882
BC00384=171115,1369889,1882
BC00385=171115,1369889,1882
BC00386=171115,1369889,1882
BC00387=171115,1369888,1879
BC00388=171115,1369888,1879
BC00389=171115,1369888,1879
BC00390=171115,1369888,1879
BC00391=171115,1369888,1879
BC00392=171115,1369888,1879
BC00393=171115,1369888,1879
BC00394=171115,1369888,1879
BC00395=171115,1369888,1879
BC00396=171115,1369888,1879
BC00397=171115,1369888,1879
BC00398=171115,1369888,1879
BC00399=171115,1369888,1879
BC00400=171115,1369888,1879
BC00401=171115,1369888,1879
BC00402=171115,1369888,1879
BC00403=171115,1369888,1879
BC00404=171115,1369887,1879
BC00405=171116,1369887,1878
BC00406=171116,1369887,1878
BC00407=171116,1369887,1878
BC00408=171116,1369887,1878
BC00409=171116,1369887,1878
BC00410=171116,1369887,1878
BC00411=171116,1369887,1878
BC00412=171116,1369887,1878
BC00413=171116,1369887,1878
BC00414=171116,1369887,1878
BC00415=171116,1369887,1878
BC00416=171116,1369887,1878
BC00417=171116,1369887,1878
BC00418=171116,1369887,1878
BC00419=171116,1369887,1878
BC00420=171116,1369887,1878
BC00421=171116,1369887,1878
BC00422=171116,1369887,1878
BC00423=171115,1369889,1882
BC00424=171115,1369889,1882
BC00425=171115,1369889,1882
BC00426=171115,1369889,1882
BC00427=171115,1369889,1882
BC00428=171115,1369889,1882
BC00429=171115,1369889,1882
BC00430=171115,1369889,1882
BC00431=171115,1369889,1882
BC00432=171115,1369889,1882
BC00433=171115,1369889,1882
BC00434=171115,1369889,1882
BC00435=171115,1369889,1882
BC00436=171115,1369889,167
BC00437=171115,1369889,167
BC00438=171115,1369889,167
BC00439=171115,1369889,167
BC00440=171115,1369889,167
BC00441=171115,1369889,167
BC00442=171115,1369889,167
BC00443=171115,1369889,167
BC00444=143530,1369889,167
BC00445=143530,1369889,167
BC00446=143530,1369889,167
BC00447=143530,1369889,167
BC00448=143530,1372986,167
BC00449=330710,1372986,167
BC00450=330710,1372986,167
BC00451=330710,1372986,167
BC00452=361518,1372956,144888
BC00453=367537,1364553,143283
BC00454=374353,1355038,141465
BC00455=398174,1321783,135113
BC00456=398174,1321783,135113
BC00457=398174,1321783,135113
BC00458=398174,1321783,135113
BC00459=398174,1321783,135110
BC00460=398174,1321783,199558
BC00461=369955,1320476,190565
BC00462=332653,1318400,176274
BC00463=350446,1306885,300644
BC00464=351050,1306811,300466
BC00465=351050,1306811,300466
BC00466=351050,1306811,300466
BC00467=351050,1306811,300466
BC00468=351050,1306811,300466
BC00469=351050,1306811,300466
BC00470=351050,1306811,300466
BC00471=351050,1306811,300466
BC00472=350446,1306885,300644
BC00473=350330,1345569,140511
BC00474=350318,1362954,38397
BC00475=350319,1362252,38395
BC00476=350318,1369188,38397
BC00477=350318,1369188,38397
BC00478=350318,1369188,38397
BC00479=350318,1369188,38393
BC00480=350318,1369188,38397
BC00481=350318,1369188,38397
BC00482=350318,1369188,38397
BC00483=350318,1369188,38397
BC00484=332907,1319511,215580
BC00485=324469,1294535,299337
BC00486=324469,1294535,299337
BC00487=324469,1294535,299337
BC00488=324469,1294535,299337
BC00489=324469,1294535,299337
BC00490=324469,1294535,299337
BC00491=324469,1294535,299337
BC00492=324469,1294535,299337
BC00493=324470,1294536,299336
BC00494=324469,1294535,299337
BC00495=324469,1294535,299337
BC00496=378057,1319426,238838
BC00497=398174,1331142,220624
BC00498=398174,1331142,220624
BC00499=398174,1331142,220624
BC00500=398174,1331142,220624
BC00501=398174,1331142,220624
BC00502=398174,1331142,220624
BC00503=398174,1331142,220624
BC00504=398174,1331142,220624
BC00505=398174,1331142,220624
BC00506=398174,1328620,215389
BC00507=359686,1333158,214696
BC00508=329122,1336762,214146
BC00509=329122,1336762,214146
BC00510=329122,1336762,214146
BC00511=329122,1336762,214146
BC00512=329122,1336762,214146
BC00513=329122,1336762,214146
BC00514=329122,1336762,214146
BC00515=329122,1336762,214146
BC00516=329122,1336762,214146
BC00517=329122,1336762,214146
BC00518=329122,1336762,214146
BC00519=329122,1336762,214146
BC00520=367015,1348719,144696
BC00521=367015,1348719,144696
BC00522=367015,1348719,144696
BC00523=367015,1348719,144696
BC00524=367015,1348719,144696
BC00525=367015,1348719,144696
BC00526=367015,1348719,144696
BC00527=367015,1348719,144696
BC00528=367015,1348719,144696
BC00529=367015,1348719,144696
BC00530=367015,1348719,144696
BC00531=346608,1354830,157578
BC00532=319155,1354830,157578
BC00533=319155,1354830,153694
BC00534=319155,1354830,153694
BC00535=319155,1354830,153694
BC00536=319155,1354830,153694
BC00537=346608,1354830,157578
BC00538=288108,1360159,194507
BC00539=269895,1363613,501241
BC00540=235813,1345575,1075229
BC00541=95044,675039,1075229
BC00542=127053,672594,1075229
EC00000=-798156,0
EC00001=-798156,0
EC00002=-798156,0
EC00003=-798156,0
EC00004=-798156,0
EC00005=-798156,0
EC00006=-798156,0
EC00007=-798156,0
EC00008=-798156,0
EC00009=-798156,0
EC00010=-798156,0
EC00011=-798156,0
EC00012=-798156,0
EC00013=-798156,0
EC00014=-798156,0
EC00015=-798156,0
EC00016=-798156,0
EC00017=-798156,0
EC00018=-798156,0
EC00019=-798156,0
EC00020=-798156,0
EC00021=-798156,0
EC00022=-798156,0
EC00023=-798156,0
EC00024=-798156,0
EC00025=-798156,0
EC00026=-798156,0
EC00027=-798156,0
EC00028=-798156,0
EC00029=-798156,0
EC00030=-798156,0
EC00031=-798156,0
EC00032=-798156,0
EC00033=-798156,0
EC00034=-798156,0
EC00035=-798156,0
EC00036=-798156,0
EC00037=-798156,0
EC00038=-798156,0
EC00039=-798156,0
EC00040=-798156,0
EC00041=-798156,0
EC00042=-798156,0
EC00043=-798156,0
EC00044=-798156,0
EC00045=-798156,0
EC00046=-798156,0
EC00047=-798156,0
EC00048=-798156,0
EC00049=-798156,0
EC00050=-798156,0
EC00051=-798156,0
EC00052=-798156,0
EC00053=-798156,0
EC00054=-798156,0
EC00055=-798156,0
EC00056=-798156,0
EC00057=-798156,0
EC00058=-798156,0
EC00059=-798156,0
EC00060=-798156,0
EC00061=-798156,0
EC00062=-798156,0
EC00063=-798156,0
EC00064=-798156,0
EC00065=-798156,0
EC00066=-798156,0
EC00067=-798156,0
EC00068=-798156,0
EC00069=-798156,0
EC00070=-798156,0
EC00071=-798156,0
EC00072=-798156,0
EC00073=-798156,0
EC00074=-798156,0
EC00075=-798156,0
EC00076=-798156,0
EC00077=-798156,0
EC00078=-798156,0
EC00079=-798156,0
EC00080=-798156,0
EC00081=-798156,0
EC00082=-798156,0
EC00083=-798156,0
EC00084=-798156,0
EC00085=-798156,0
EC00086=-798156,0
EC00087=-798156,0
EC00088=-798156,0
EC00089=-798156,0
EC00090=-798156,0
EC00091=-798156,0
EC00092=-798156,0
EC00093=-798156,0
EC00094=-798156,0
EC00095=-798156,0
EC00096=-798156,0
EC00097=-798156,0
EC00098=-798156,0
EC00099=-798156,0
EC00100=-798156,0
EC00101=-798156,0
EC00102=-798156,0
EC00103=-798156,0
EC00104=-798156,0
EC00105=-798156,0
EC00106=-798156,0
EC00107=-798156,0
EC00108=-798156,0
EC00109=-798156,0
EC00110=-798156,0
EC00111=-798156,0
EC00112=-798156,0
EC00113=-798156,0
EC00114=-798156,0
EC00115=-798156,0
EC00116=-798156,0
EC00117=-798156,0
EC00118=-798156,0
EC00119=-798156,0
EC00120=-798156,0
EC00121=-798156,0
EC00122=-798156,0
EC00123=-798156,0
EC00124=-798156,0
EC00125=-798156,0
EC00126=-798156,0
EC00127=-798156,0
EC00128=-798156,0
EC00129=-798156,0
EC00130=-798156,0
EC00131=-798156,0
EC00132=-798156,0
EC00133=-798156,0
EC00134=-798156,0
EC00135=-798156,0
EC00136=-798156,0
EC00137=-798156,0
EC00138=-798156,0
EC00139=-798156,0
EC00140=-798156,0
EC00141=-798156,0
EC00142=-798156,0
EC00143=-798156,0
EC00144=-798156,0
EC00145=-798156,0
EC00146=-798156,0
EC00147=-798156,0
EC00148=-798156,0
EC00149=-798156,0
EC00150=-798156,0
EC00151=-798156,0
EC00152=-798156,0
EC00153=-798156,0
EC00154=-798156,0
EC00155=-798156,0
EC00156=-798156,0
EC00157=-798156,0
EC00158=-798156,0
EC00159=-798156,0
EC00160=-798156,0
EC00161=-798156,0
EC00162=-798156,0
EC00163=-798156,0
EC00164=-798156,0
EC00165=-798156,0
EC00166=-798156,0
EC00167=-798156,0
EC00168=-798156,0
EC00169=-798156,0
EC00170=-798156,0
EC00171=-798156,0
EC00172=-798156,0
EC00173=-798156,0
EC00174=-798156,0
EC00175=-798156,0
EC00176=-798156,0
EC00177=-798156,0
EC00178=-798156,0
EC00179=-798156,0
EC00180=-798156,0
EC00181=-798156,0
EC00182=-798156,0
EC00183=-798156,0
EC00184=-798156,0
EC00185=-798156,0
EC00186=-798156,0
EC00187=-798156,0
EC00188=-798156,0
EC00189=-798156,0
EC00190=-798156,0
EC00191=-798156,0
EC00192=-798156,0
EC00193=-798156,0
EC00194=-798156,0
EC00195=-798156,0
EC00196=-798156,0
EC00197=-798156,0
EC00198=-798156,0
EC00199=-798156,0
EC00200=-798156,0
EC00201=-798156,0
EC00202=-798156,0
EC00203=-798156,0
EC00204=-798156,0
EC00205=-798156,0
EC00206=-798156,0
EC00207=-798156,0
EC00208=-798156,0
EC00209=-798155,0
EC00210=-798155,0
EC00211=-798155,0
EC00212=-798155,0
EC00213=-798155,0
EC00214=-798156,0
EC00215=-798156,0
EC00216=-798156,0
EC00217=-798156,0
EC00218=-798156,0
EC00219=-798156,0
EC00220=-798156,0
EC00221=-798155,-1
EC00222=-798156,0
EC00223=-798156,0
EC00224=-798156,0
EC00225=-798156,0
EC00226=-798156,0
EC00227=-798156,0
EC00228=-798156,0
EC00229=-798156,0
EC00230=-798156,0
EC00231=-798156,0
EC00232=-798156,0
EC00233=-798156,0
EC00234=-798156,0
EC00235=-798156,0
EC00236=-798156,0
EC00237=-798156,0
EC00238=-798156,0
EC00239=-798156,0
EC00240=-798156,0
EC00241=-798156,0
EC00242=-798156,0
EC00243=-798156,0
EC00244=-798156,0
EC00245=-798156,0
EC00246=-798156,0
EC00247=-798156,0
EC00248=-798156,0
EC00249=-798156,0
EC00250=-798156,0
EC00251=-798156,0
EC00252=-798156,0
EC00253=-798156,0
EC00254=-798156,0
EC00255=-798156,0
EC00256=-798156,0
EC00257=-798156,0
EC00258=-798156,0
EC00259=-798156,0
EC00260=-798156,0
EC00261=-798156,0
EC00262=-798156,0
EC00263=-798156,0
EC00264=-798156,0
EC00265=-798156,0
EC00266=-798156,0
EC00267=-798156,0
EC00268=-798156,0
EC00269=-798156,0
EC00270=-798156,0
EC00271=-798156,0
EC00272=-798156,0
EC00273=-798156,0
EC00274=-798156,0
EC00275=-798156,0
EC00276=-798156,0
EC00277=-798156,0
EC00278=-798156,0
EC00279=-798156,0
EC00280=-798156,0
EC00281=-798156,0
EC00282=-798156,0
EC00283=-798156,0
EC00284=-798156,0
EC00285=-798156,0
EC00286=-798156,0
EC00287=-798156,0
EC00288=-798156,0
EC00289=-798156,0
EC00290=798156,0
EC00291=798156,0
EC00292=798156,0
EC00293=798156,0
EC00294=798156,0
EC00295=798156,0
EC00296=798156,0
EC00297=798156,0
EC00298=798156,0
EC00299=798156,0
EC00300=798156,0
EC00301=798156,0
EC00302=798156,0
EC00303=798156,0
EC00304=798156,0
EC00305=798156,0
EC00306=798156,0
EC00307=798156,0
EC00308=798156,0
EC00309=798156,0
EC00310=798156,0
EC00311=798156,0
EC00312=798156,0
EC00313=798156,0
EC00314=798156,0
EC00315=798156,0
EC00316=798156,0
EC00317=798156,0
EC00318=798156,0
EC00319=798156,0
EC00320=798156,0
EC00321=798156,0
EC00322=798156,0
EC00323=798156,0
EC00324=798156,0
EC00325=798156,0
EC00326=798156,0
EC00327=798156,0
EC00328=798156,0
EC00329=798156,0
EC00330=798156,0
EC00331=798156,0
EC00332=798156,0
EC00333=798156,0
EC00334=798156,0
EC00335=798156,0
EC00336=798156,0
EC00337=798156,0
EC00338=798156,0
EC00339=798156,0
EC00340=798156,0
EC00341=798156,0
EC00342=798156,0
EC00343=798156,0
EC00344=798156,0
EC00345=798156,0
EC00346=798156,0
EC00347=798156,0
EC00348=798156,0
EC00349=798156,0
EC00350=798156,0
EC00351=798156,0
EC00352=798156,0
EC00353=798156,0
EC00354=798156,0
EC00355=798156,0
EC00356=798156,0
EC00357=798156,0
EC00358=798156,0
EC00359=798156,0
EC00360=798156,0
EC00361=798156,0
EC00362=798156,0
EC00363=798156,0
EC00364=798156,0
EC00365=798156,0
EC00366=798156,0
EC00367=798156,0
EC00368=798156,0
EC00369=798156,0
EC00370=798156,0
EC00371=798156,0
EC00372=798156,0
EC00373=798155,0
EC00374=798155,0
EC00375=798155,0
EC00376=798155,0
EC00377=798155,0
EC00378=798155,0
EC00379=798155,0
EC00380=798155,0
EC00381=798155,0
EC00382=798155,0
EC00383=798155,0
EC00384=798155,0
EC00385=798155,0
EC00386=798155,0
EC00387=798155,1
EC00388=798155,1
EC00389=798155,1
EC00390=798155,1
EC00391=798155,1
EC00392=798155,1
EC00393=798155,1
EC00394=798155,1
EC00395=798155,1
EC00396=798155,1
EC00397=798155,1
EC00398=798155,1
EC00399=798155,1
EC00400=798155,1
EC00401=798155,1
EC00402=798155,1
EC00403=798155,1
EC00404=798154,1
EC00405=798153,2
EC00406=798153,2
EC00407=798153,2
EC00408=798153,2
EC00409=798153,2
EC00410=798153,2
EC00411=798153,2
EC00412=798153,2
EC00413=798153,2
EC00414=798153,2
EC00415=798153,2
EC00416=798153,2
EC00417=798153,2
EC00418=798153,2
EC00419=798153,2
EC00420=798153,2
EC00421=798153,2
EC00422=798153,2
EC00423=798155,0
EC00424=798155,0
EC00425=798155,0
EC00426=798155,0
EC00427=798155,0
EC00428=798155,0
EC00429=798155,0
EC00430=798155,0
EC00431=798155,0
EC00432=798155,0
EC00433=798155,0
EC00434=798155,0
EC00435=798155,0
EC00436=798155,0
EC00437=798155,0
EC00438=798155,0
EC00439=798155,0
EC00440=798155,0
EC00441=798155,0
EC00442=798155,0
EC00443=798155,0
EC00444=798155,0
EC00445=798155,0
EC00446=798155,0
EC00447=798155,0
EC00448=798155,0
EC00449=798155,0
EC00450=798155,0
EC00451=798155,0
EC00452=798156,0
EC00453=798156,0
EC00454=798156,0
EC00455=798156,0
EC00456=798156,0
EC00457=798156,0
EC00458=798156,0
EC00459=798155,1
EC00460=798155,1
EC00461=798155,1
EC00462=798156,0
EC00463=798156,0
EC00464=798156,0
EC00465=798156,0
EC00466=798156,0
EC00467=798156,0
EC00468=798156,0
EC00469=798156,0
EC00470=798156,0
EC00471=798156,0
EC00472=798156,0
EC00473=798156,0
EC00474=798156,0
EC00475=798155,0
EC00476=798156,0
EC00477=798156,0
EC00478=798156,0
EC00479=798155,1
EC00480=798156,0
EC00481=798156,0
EC00482=798156,0
EC00483=798156,0
EC00484=798156,0
EC00485=798156,0
EC00486=798156,0
EC00487=798156,0
EC00488=798156,0
EC00489=798156,0
EC00490=798156,0
EC00491=798156,0
EC00492=798156,0
EC00493=798155,1
EC00494=798156,0
EC00495=798156,0
EC00496=798156,0
EC00497=798156,0
EC00498=798156,0
EC00499=798156,0
EC00500=798156,0
EC00501=798156,0
EC00502=798156,0
EC00503=798156,0
EC00504=798156,0
EC00505=798156,0
EC00506=798156,0
EC00507=798156,0
EC00508=798156,0
EC00509=798156,0
EC00510=798156,0
EC00511=798156,0
EC00512=798156,0
EC00513=798156,0
EC00514=798156,0
EC00515=798156,0
EC00516=798156,0
EC00517=798156,0
EC00518=798156,0
EC00519=798156,0
EC00520=798156,0
EC00521=798156,0
EC00522=798156,0
EC00523=798156,0
EC00524=798156,0
EC00525=798156,0
EC00526=798156,0
EC00527=798156,0
EC00528=798156,0
EC00529=798156,0
EC00530=798156,0
EC00531=798156,0
EC00532=798156,0
EC00533=798156,0
EC00534=798156,0
EC00535=798156,0
EC00536=798156,0
EC00537=798156,0
EC00538=798156,0
EC00539=798156,0
EC00540=798156,0
EC00541=798156,0
EC00542=798156,0
///POSTYPE BASE
///RECTAN
///RCONF 0,0,0,0,0,0,0,0,0,0,0,0,0,0,0,0,0,0,0,0,0,0,0,0
P00006=0.222,-3.123,-1.508,0.0000,0.0000,0.0000
P00021=-0.225,-6.128,-0.405,0.0000,0.0000,0.0000
P00022=0.222,-3.123,-1.508,0.0000,0.0000,0.0000
P00023=0.143,-0.036,0.682,0.0000,0.0000,0.0000
P00024=0.145,-0.552,1.326,0.0000,0.0000,0.0000
P00025=-2.003,0.006,0.728,0.0000,0.0000,0.0000
P00026=0.562,-0.002,-0.337,0.0000,0.0000,0.0000
P00027=-0.746,0.015,-9.096,0.0000,0.0000,0.0000
P00031=1.853,-0.001,-1.549,0.0000,0.0000,0.0000
P00050=4.296,-4.501,-0.826,0.0000,0.0000,0.0000
P00051=0.367,3.892,0.009,0.0000,0.0000,0.0000
P00052=0.088,2.832,-0.342,0.0000,0.0000,0.0000
P00053=0.134,6.594,0.107,0.0000,0.0000,0.0000
P00054=-0.103,6.509,-0.702,0.0000,0.0000,0.0000
P00055=-0.342,8.912,1.324,0.0000,0.0000,0.0000
//INST
///DATE 2025/05/19 13:35
///ATTR SC,RW
///GROUP1 RB1,BS1
///GROUP2 ST1
NOP
'POPRAWIC POM DODAC HARDOXY
'X2_34-37(-90,0)
'210,0
MOVJ C00000 BC00000 VJ=100.00  +MOVJ EC00000 VJ=100.00
'Path S3633
SFTOF3D
MOVJ C00001 BC00001 VJ=100.00  +MOVJ EC00001 VJ=100.00
MOVL C00002 BC00002 V=800.0  +MOVJ EC00002 VJ=100.00
SMOVL C00003 BC00003 V=166.7  +MOVJ EC00003
SREFP 3 C00004 BC00004  +REFP EC00004
CALL JOB:SEARCH-R1-S13D
SET P021 P006
SFTON3D P021
SMOVL C00005 BC00005 V=166.7  +MOVJ EC00005
SREFP 3 C00006 BC00006  +REFP EC00006
CALL JOB:SEARCH-R1-S13D
SET P021 P006
SFTON3D P021
SMOVL C00007 BC00007 V=166.7  +MOVJ EC00007
SMOVL C00008 BC00008 V=166.7  +MOVJ EC00008
SREFP 3 C00009 BC00009  +REFP EC00009
CALL JOB:SEARCH-R1-S13D
SET P021 P006
SFTON3D P021
SMOVL C00010 BC00010 V=166.7  +MOVJ EC00010
SFTOF3D
SMOVL C00011 BC00011 V=250.0  +MOVJ EC00011
SMOVL C00012 BC00012 V=166.7  +MOVJ EC00012
SREFP 3 C00013 BC00013  +REFP EC00013
CALL JOB:SEARCH-R1-S13D
SET P031 P006
SFTON3D P031
SMOVL C00014 BC00014 V=166.7  +MOVJ EC00014
SREFP 3 C00015 BC00015  +REFP EC00015
CALL JOB:SEARCH-R1-S13D
SET P031 P006
SFTON3D P031
SMOVL C00016 BC00016 V=166.7  +MOVJ EC00016
MOVL C00017 BC00017 V=800.0  +MOVJ EC00017 VJ=100.00
MOVL C00018 BC00018 V=1000.0  +MOVJ EC00018 VJ=100.00
'EndPath S3633
'Path S4258
SFTOF3D
MOVJ C00019 BC00019 VJ=100.00  +MOVJ EC00019 VJ=100.00
MOVL C00020 BC00020 V=800.0  +MOVJ EC00020 VJ=100.00
SMOVL C00021 BC00021 V=166.7  +MOVJ EC00021
SREFP 3 C00022 BC00022  +REFP EC00022
CALL JOB:SEARCH-R1-S13D
SET P022 P006
SFTON3D P022
SMOVL C00023 BC00023 V=166.7  +MOVJ EC00023
SMOVL C00024 BC00024 V=166.7  +MOVJ EC00024
SREFP 3 C00025 BC00025  +REFP EC00025
CALL JOB:SEARCH-R1-S13D
SET P022 P006
SFTON3D P022
SMOVL C00026 BC00026 V=166.7  +MOVJ EC00026
SMOVL C00027 BC00027 V=166.7  +MOVJ EC00027
SMOVL C00028 BC00028 V=166.7  +MOVJ EC00028
SREFP 3 C00029 BC00029  +REFP EC00029
CALL JOB:SEARCH-R1-S13D
SET P022 P006
SFTON3D P022
SMOVL C00030 BC00030 V=166.7  +MOVJ EC00030
SMOVL C00031 BC00031 V=166.7  +MOVJ EC00031
SMOVL C00032 BC00032 V=166.7  +MOVJ EC00032
MOVL C00033 BC00033 V=800.0  +MOVJ EC00033 VJ=100.00
MOVL C00034 BC00034 V=1000.0  +MOVJ EC00034 VJ=100.00
'EndPath S4258
'Path S4259
SFTOF3D
MOVJ C00035 BC00035 VJ=100.00  +MOVJ EC00035 VJ=100.00
MOVL C00036 BC00036 V=800.0  +MOVJ EC00036 VJ=100.00
SMOVL C00037 BC00037 V=166.7  +MOVJ EC00037
SREFP 3 C00038 BC00038  +REFP EC00038
CALL JOB:SEARCH-R1-S13D
SET P023 P006
SFTON3D P023
SMOVL C00039 BC00039 V=166.7  +MOVJ EC00039
SMOVL C00040 BC00040 V=166.7  +MOVJ EC00040
SREFP 3 C00041 BC00041  +REFP EC00041
CALL JOB:SEARCH-R1-S13D
SET P023 P006
SFTON3D P023
SMOVL C00042 BC00042 V=166.7  +MOVJ EC00042
SMOVL C00043 BC00043 V=166.7  +MOVJ EC00043
SREFP 3 C00044 BC00044  +REFP EC00044
CALL JOB:SEARCH-R1-S13D
SET P023 P006
SFTON3D P023
SMOVL C00045 BC00045 V=166.7  +MOVJ EC00045
MOVL C00046 BC00046 V=800.0  +MOVJ EC00046 VJ=100.00
MOVL C00047 BC00047 V=1000.0  +MOVJ EC00047 VJ=100.00
'EndPath S4259
'Path S4260
SFTOF3D
MOVJ C00048 BC00048 VJ=100.00  +MOVJ EC00048 VJ=100.00
MOVL C00049 BC00049 V=800.0  +MOVJ EC00049 VJ=100.00
SMOVL C00050 BC00050 V=166.7  +MOVJ EC00050
SREFP 3 C00051 BC00051  +REFP EC00051
CALL JOB:SEARCH-R1-S13D
SET P024 P006
SFTON3D P024
SMOVL C00052 BC00052 V=166.7  +MOVJ EC00052
SMOVL C00053 BC00053 V=166.7  +MOVJ EC00053
SREFP 3 C00054 BC00054  +REFP EC00054
CALL JOB:SEARCH-R1-S13D
SET P024 P006
SFTON3D P024
SMOVL C00055 BC00055 V=166.7  +MOVJ EC00055
SMOVL C00056 BC00056 V=166.7  +MOVJ EC00056
SMOVL C00057 BC00057 V=166.7  +MOVJ EC00057
SREFP 3 C00058 BC00058  +REFP EC00058
CALL JOB:SEARCH-R1-S13D
SET P024 P006
SFTON3D P024
SMOVL C00059 BC00059 V=166.7  +MOVJ EC00059
SMOVL C00060 BC00060 V=166.7  +MOVJ EC00060
MOVL C00061 BC00061 V=1000.0  +MOVJ EC00061 VJ=100.00
'EndPath S4260
'Path S4261
SFTOF3D
MOVJ C00062 BC00062 VJ=100.00  +MOVJ EC00062 VJ=100.00
MOVL C00063 BC00063 V=800.0  +MOVJ EC00063 VJ=100.00
SMOVL C00064 BC00064 V=166.7  +MOVJ EC00064
SREFP 3 C00065 BC00065  +REFP EC00065
CALL JOB:SEARCH-R1-S13D
SET P025 P006
SFTON3D P025
SMOVL C00066 BC00066 V=166.7  +MOVJ EC00066
SMOVL C00067 BC00067 V=166.7  +MOVJ EC00067
SREFP 3 C00068 BC00068  +REFP EC00068
CALL JOB:SEARCH-R1-S13D
SET P025 P006
SFTON3D P025
SMOVL C00069 BC00069 V=166.7  +MOVJ EC00069
SMOVL C00070 BC00070 V=166.7  +MOVJ EC00070
SREFP 3 C00071 BC00071  +REFP EC00071
CALL JOB:SEARCH-R1-S13D
SET P025 P006
SFTON3D P025
SMOVL C00072 BC00072 V=166.7  +MOVJ EC00072
MOVL C00073 BC00073 V=1000.0  +MOVJ EC00073 VJ=100.00
'EndPath S4261
'Path S4262
SFTOF3D
MOVJ C00074 BC00074 VJ=100.00  +MOVJ EC00074 VJ=100.00
MOVL C00075 BC00075 V=800.0  +MOVJ EC00075 VJ=100.00
SMOVL C00076 BC00076 V=166.7  +MOVJ EC00076
SREFP 3 C00077 BC00077  +REFP EC00077
CALL JOB:SEARCH-R1-S13D
SET P026 P006
SFTON3D P026
SMOVL C00078 BC00078 V=166.7  +MOVJ EC00078
SMOVL C00079 BC00079 V=166.7  +MOVJ EC00079
SREFP 3 C00080 BC00080  +REFP EC00080
CALL JOB:SEARCH-R1-S13D
SET P026 P006
SFTON3D P026
SMOVL C00081 BC00081 V=166.7  +MOVJ EC00081
SMOVL C00082 BC00082 V=166.7  +MOVJ EC00082
SMOVL C00083 BC00083 V=166.7  +MOVJ EC00083
SREFP 3 C00084 BC00084  +REFP EC00084
CALL JOB:SEARCH-R1-S13D
SET P026 P006
SFTON3D P026
SMOVL C00085 BC00085 V=166.7  +MOVJ EC00085
MOVL C00086 BC00086 V=1000.0  +MOVJ EC00086 VJ=100.00
'EndPath S4262
'Path S4263
SFTOF3D
MOVJ C00087 BC00087 VJ=100.00  +MOVJ EC00087 VJ=100.00
MOVL C00088 BC00088 V=800.0  +MOVJ EC00088 VJ=100.00
SMOVL C00089 BC00089 V=166.7  +MOVJ EC00089
SREFP 3 C00090 BC00090  +REFP EC00090
CALL JOB:SEARCH-R1-S13D
SET P027 P006
SFTON3D P027
SMOVL C00091 BC00091 V=166.7  +MOVJ EC00091
SMOVL C00092 BC00092 V=166.7  +MOVJ EC00092
SREFP 3 C00093 BC00093  +REFP EC00093
CALL JOB:SEARCH-R1-S13D
SET P027 P006
SFTON3D P027
SMOVL C00094 BC00094 V=166.7  +MOVJ EC00094
SMOVL C00095 BC00095 V=166.7  +MOVJ EC00095
SMOVL C00096 BC00096 V=166.7  +MOVJ EC00096
SREFP 3 C00097 BC00097  +REFP EC00097
CALL JOB:SEARCH-R1-S13D
SET P027 P006
SFTON3D P027
SMOVL C00098 BC00098 V=166.7  +MOVJ EC00098
SMOVL C00099 BC00099 V=166.7  +MOVJ EC00099
SMOVL C00100 BC00100 V=166.7  +MOVJ EC00100
MOVL C00101 BC00101 V=800.0  +MOVJ EC00101 VJ=100.00
MOVL C00102 BC00102 V=1000.0  +MOVJ EC00102 VJ=100.00
SFTOF3D
MOVL C00103 BC00103 V=1000.0  +MOVJ EC00103 VJ=100.00
MOVL C00104 BC00104 V=1000.0  +MOVJ EC00104 VJ=100.00
SMOVL C00105 BC00105 V=166.7  +MOVJ EC00105
SREFP 3 C00106 BC00106  +REFP EC00106
CALL JOB:SEARCH-R1-S13D
SET P051 P006
SFTON3D P051
SMOVL C00107 BC00107 V=166.7  +MOVJ EC00107
SREFP 3 C00108 BC00108  +REFP EC00108
CALL JOB:SEARCH-R1-S13D
SET P051 P006
SFTON3D P051
SMOVL C00109 BC00109 V=166.7  +MOVJ EC00109
SFTOF3D
MOVL C00110 BC00110 V=1000.0  +MOVJ EC00110 VJ=100.00
MOVL C00111 BC00111 V=1000.0  +MOVJ EC00111 VJ=100.00
SMOVL C00112 BC00112 V=166.7  +MOVJ EC00112
SREFP 3 C00113 BC00113  +REFP EC00113
CALL JOB:SEARCH-R1-S13D
SET P050 P006
SFTON3D P050
SMOVL C00114 BC00114 V=166.7  +MOVJ EC00114
SREFP 3 C00115 BC00115  +REFP EC00115
CALL JOB:SEARCH-R1-S13D
SET P050 P006
SFTON3D P050
SMOVL C00116 BC00116 V=166.7  +MOVJ EC00116
SFTOF3D
MOVL C00117 BC00117 V=1000.0  +MOVJ EC00117 VJ=100.00
MOVL C00118 BC00118 V=1000.0  +MOVJ EC00118 VJ=100.00
MOVL C00119 BC00119 V=1000.0  +MOVJ EC00119 VJ=100.00
MOVL C00120 BC00120 V=1000.0  +MOVJ EC00120 VJ=100.00
MOVL C00121 BC00121 V=1000.0  +MOVJ EC00121 VJ=100.00
MOVL C00122 BC00122 V=1000.0  +MOVJ EC00122 VJ=100.00
SFTOF3D
MOVL C00123 BC00123 V=1000.0  +MOVJ EC00123 VJ=100.00
SMOVL C00124 BC00124 V=166.7  +MOVJ EC00124
SREFP 3 C00125 BC00125  +REFP EC00125
CALL JOB:SEARCH-R1-S13D
SET P053 P006
SFTON3D P053
SMOVL C00126 BC00126 V=166.7  +MOVJ EC00126
SREFP 3 C00127 BC00127  +REFP EC00127
CALL JOB:SEARCH-R1-S13D
SET P053 P006
SFTON3D P053
SMOVL C00128 BC00128 V=166.7  +MOVJ EC00128
SMOVL C00129 BC00129 V=166.7  +MOVJ EC00129
SMOVL C00130 BC00130 V=166.7  +MOVJ EC00130
SREFP 3 C00131 BC00131  +REFP EC00131
CALL JOB:SEARCH-R1-S13D
SET P053 P006
SFTON3D P053
SMOVL C00132 BC00132 V=166.7  +MOVJ EC00132
SMOVL C00133 BC00133 V=166.7  +MOVJ EC00133
SMOVL C00134 BC00134 V=166.7  +MOVJ EC00134
SREFP 3 C00135 BC00135  +REFP EC00135
CALL JOB:SEARCH-R1-S13D
SET P053 P006
SFTON3D P053
SMOVL C00136 BC00136 V=166.7  +MOVJ EC00136
SFTOF3D
MOVL C00137 BC00137 V=1000.0  +MOVJ EC00137 VJ=100.00
MOVL C00138 BC00138 V=1000.0  +MOVJ EC00138 VJ=100.00
SMOVL C00139 BC00139 V=166.7  +MOVJ EC00139
SREFP 3 C00140 BC00140  +REFP EC00140
CALL JOB:SEARCH-R1-S13D
SET P052 P006
SFTON3D P052
SMOVL C00141 BC00141 V=166.7  +MOVJ EC00141
SREFP 3 C00142 BC00142  +REFP EC00142
CALL JOB:SEARCH-R1-S13D
SET P052 P006
SFTON3D P052
SMOVL C00143 BC00143 V=166.7  +MOVJ EC00143
SFTOF3D
MOVL C00144 BC00144 V=1000.0  +MOVJ EC00144 VJ=100.00
MOVL C00145 BC00145 V=1000.0  +MOVJ EC00145 VJ=100.00
MOVL C00146 BC00146 V=1000.0  +MOVJ EC00146 VJ=100.00
SMOVL C00147 BC00147 V=166.7  +MOVJ EC00147
SREFP 3 C00148 BC00148  +REFP EC00148
CALL JOB:SEARCH-R1-S13D
SET P054 P006
SFTON3D P054
SMOVL C00149 BC00149 V=166.7  +MOVJ EC00149
SMOVL C00150 BC00150 V=166.7  +MOVJ EC00150
SMOVL C00151 BC00151 V=166.7  +MOVJ EC00151
SREFP 3 C00152 BC00152  +REFP EC00152
CALL JOB:SEARCH-R1-S13D
SET P054 P006
SFTON3D P054
SMOVL C00153 BC00153 V=166.7  +MOVJ EC00153
SMOVL C00154 BC00154 V=166.7  +MOVJ EC00154
SMOVL C00155 BC00155 V=166.7  +MOVJ EC00155
SREFP 3 C00156 BC00156  +REFP EC00156
CALL JOB:SEARCH-R1-S13D
SET P054 P006
SFTON3D P054
SMOVL C00157 BC00157 V=166.7  +MOVJ EC00157
SFTOF3D
MOVL C00158 BC00158 V=1000.0  +MOVJ EC00158 VJ=100.00
SMOVL C00159 BC00159 V=166.7  +MOVJ EC00159
SREFP 3 C00160 BC00160  +REFP EC00160
CALL JOB:SEARCH-R1-S13D
SET P055 P006
SFTON3D P055
SMOVL C00161 BC00161 V=166.7  +MOVJ EC00161
SREFP 3 C00162 BC00162  +REFP EC00162
CALL JOB:SEARCH-R1-S13D
SET P055 P006
SFTON3D P055
SMOVL C00163 BC00163 V=166.7  +MOVJ EC00163
SFTOF3D
MOVL C00164 BC00164 V=1000.0  +MOVJ EC00164 VJ=100.00
SFTON3D P054
SMOVL C00165 BC00165 V=150.0 PL=0  +MOVJ EC00165
MACRO1 MJ#(0) ARGF9
ARCON
SMOVL C00166 BC00166 V=10.0  +MOVJ EC00166
SMOVC C00167 BC00167 V=13.3  +MOVJ EC00167
SMOVC C00168 BC00168 V=13.3  +MOVJ EC00168
SMOVC C00169 BC00169 V=13.3  +MOVJ EC00169
SMOVL C00170 BC00170 V=10.0  +MOVJ EC00170
SFTON3D P055
SMOVL C00171 BC00171 V=10.0  +MOVJ EC00171
ARCOF
SMOVL C00172 BC00172 V=166.7  +MOVJ EC00172
SFTOF3D
SMOVL C00173 BC00173 V=333.3  +MOVJ EC00173
SMOVL C00174 BC00174 V=333.3  +MOVJ EC00174
SFTON3D P053
SMOVL C00175 BC00175 V=150.0 PL=0  +MOVJ EC00175
MACRO1 MJ#(0) ARGF9
ARCON
SMOVL C00176 BC00176 V=10.0  +MOVJ EC00176
SMOVC C00177 BC00177 V=13.3  +MOVJ EC00177
SMOVC C00178 BC00178 V=13.3  +MOVJ EC00178
SMOVC C00179 BC00179 V=13.3  +MOVJ EC00179
SMOVL C00180 BC00180 V=11.7  +MOVJ EC00180
SFTON3D P052
SMOVL C00181 BC00181 V=11.7  +MOVJ EC00181
SMOVL C00182 BC00182 V=11.7  +MOVJ EC00182
ARCOF
SMOVL C00183 BC00183 V=166.7  +MOVJ EC00183
SFTOF3D
MOVL C00184 BC00184 V=1000.0  +MOVJ EC00184 VJ=100.00
MOVL C00185 BC00185 V=1000.0  +MOVJ EC00185 VJ=100.00
MOVL C00186 BC00186 V=1000.0  +MOVJ EC00186 VJ=100.00
MOVL C00187 BC00187 V=1000.0  +MOVJ EC00187 VJ=100.00
MOVJ C00188 BC00188 VJ=100.00  +MOVJ EC00188 VJ=100.00
'EndPath S4263
'
'Path W4264
SFTOF3D
MOVJ C00189 BC00189 VJ=100.00  +MOVJ EC00189 VJ=100.00
MOVJ C00190 BC00190 VJ=100.00  +MOVJ EC00190 VJ=100.00
MOVJ C00191 BC00191 VJ=100.00  +MOVJ EC00191 VJ=100.00
SFTON3D P027
MOVJ C00192 BC00192 VJ=100.00  +MOVJ EC00192 VJ=100.00
MOVJ C00193 BC00193 VJ=100.00  +MOVJ EC00193 VJ=100.00
SMOVL C00194 BC00194 V=800.0  +MOVJ EC00194
SMOVL C00195 BC00195 V=150.0 PL=0  +MOVJ EC00195
MACRO1 MJ#(0) ARGF9
ARCON
SMOVL C00196 BC00196 V=10.0  +MOVJ EC00196
SMOVL C00197 BC00197 V=10.0  +MOVJ EC00197
SMOVL C00198 BC00198 V=7.5  +MOVJ EC00198
SMOVL C00199 BC00199 V=10.0  +MOVJ EC00199
ARCOF
SMOVL C00200 BC00200 V=800.0  +MOVJ EC00200
SMOVL C00201 BC00201 V=1000.0  +MOVJ EC00201
SFTOF3D
'EndPath W4264
MOVJ C00202 BC00202 VJ=100.00  +MOVJ EC00202 VJ=100.00
MOVJ C00203 BC00203 VJ=100.00  +MOVJ EC00203 VJ=100.00
MOVJ C00204 BC00204 VJ=100.00  +MOVJ EC00204 VJ=100.00
'Path W4265
SFTOF3D
SFTON3D P021
MOVJ C00205 BC00205 VJ=100.00  +MOVJ EC00205 VJ=100.00
SMOVL C00206 BC00206 V=800.0  +MOVJ EC00206
SMOVL C00207 BC00207 V=150.0 PL=0  +MOVJ EC00207
ARCON
SMOVL C00208 BC00208 V=10.0  +MOVJ EC00208
SMOVL C00209 BC00209 V=7.5  +MOVJ EC00209
SMOVL C00210 BC00210 V=7.5  +MOVJ EC00210
SFTON3D P031
SMOVL C00211 BC00211 V=9.2  +MOVJ EC00211
SMOVL C00212 BC00212 V=9.2  +MOVJ EC00212
ARCOF
SMOVL C00213 BC00213 V=250.0  +MOVJ EC00213
SMOVL C00214 BC00214 V=800.0  +MOVJ EC00214
SMOVL C00215 BC00215 V=1000.0  +MOVJ EC00215
SFTOF3D
'EndPath W4265
MOVJ C00216 BC00216 VJ=100.00  +MOVJ EC00216 VJ=100.00
MOVJ C00217 BC00217 VJ=100.00  +MOVJ EC00217 VJ=100.00
MOVJ C00218 BC00218 VJ=100.00  +MOVJ EC00218 VJ=100.00
'Path W4266
SFTOF3D
SFTON3D P025
MOVJ C00219 BC00219 VJ=100.00  +MOVJ EC00219 VJ=100.00
SMOVL C00220 BC00220 V=800.0  +MOVJ EC00220
SMOVL C00221 BC00221 V=150.0 PL=0  +MOVJ EC00221
ARCON
SMOVL C00222 BC00222 V=9.2  +MOVJ EC00222
SMOVL C00223 BC00223 V=9.2  +MOVJ EC00223
SMOVL C00224 BC00224 V=10.0  +MOVJ EC00224
SMOVL C00225 BC00225 V=9.2  +MOVJ EC00225
SMOVL C00226 BC00226 V=9.2  +MOVJ EC00226
SMOVL C00227 BC00227 V=9.2  +MOVJ EC00227
ARCOF
SMOVL C00228 BC00228 V=800.0  +MOVJ EC00228
SMOVL C00229 BC00229 V=1000.0  +MOVJ EC00229
SFTOF3D
'EndPath W4266
MOVJ C00230 BC00230 VJ=100.00  +MOVJ EC00230 VJ=100.00
MOVJ C00231 BC00231 VJ=100.00  +MOVJ EC00231 VJ=100.00
MOVJ C00232 BC00232 VJ=100.00  +MOVJ EC00232 VJ=100.00
'Path W4267
SFTOF3D
SFTON3D P023
MOVJ C00233 BC00233 VJ=100.00  +MOVJ EC00233 VJ=100.00
SMOVL C00234 BC00234 V=800.0  +MOVJ EC00234
SMOVL C00235 BC00235 V=150.0 PL=0  +MOVJ EC00235
ARCON
SMOVL C00236 BC00236 V=9.2  +MOVJ EC00236
SMOVL C00237 BC00237 V=9.2  +MOVJ EC00237
SMOVL C00238 BC00238 V=9.2  +MOVJ EC00238
SMOVL C00239 BC00239 V=9.2  +MOVJ EC00239
ARCOF
SMOVL C00240 BC00240 V=800.0  +MOVJ EC00240
SMOVL C00241 BC00241 V=1000.0  +MOVJ EC00241
SFTOF3D
'EndPath W4267
MOVJ C00242 BC00242 VJ=100.00  +MOVJ EC00242 VJ=100.00
MOVJ C00243 BC00243 VJ=100.00  +MOVJ EC00243 VJ=100.00
'
'Path W4268
SFTOF3D
SFTON3D P026
MOVJ C00244 BC00244 VJ=100.00  +MOVJ EC00244 VJ=100.00
SMOVL C00245 BC00245 V=800.0  +MOVJ EC00245
SMOVL C00246 BC00246 V=150.0 PL=0  +MOVJ EC00246
ARCON
SMOVL C00247 BC00247 V=9.2  +MOVJ EC00247
SMOVL C00248 BC00248 V=9.2  +MOVJ EC00248
SMOVL C00249 BC00249 V=9.2  +MOVJ EC00249
SMOVL C00250 BC00250 V=9.2  +MOVJ EC00250
ARCOF
SMOVL C00251 BC00251 V=800.0  +MOVJ EC00251
SMOVL C00252 BC00252 V=1000.0  +MOVJ EC00252
SFTOF3D
'EndPath W4268
MOVJ C00253 BC00253 VJ=100.00  +MOVJ EC00253 VJ=100.00
MOVJ C00254 BC00254 VJ=100.00  +MOVJ EC00254 VJ=100.00
MOVJ C00255 BC00255 VJ=100.00  +MOVJ EC00255 VJ=100.00
'Path W3636
SFTOF3D
SFTON3D P022
MOVJ C00256 BC00256 VJ=100.00  +MOVJ EC00256 VJ=100.00
SMOVL C00257 BC00257 V=800.0  +MOVJ EC00257
SMOVL C00258 BC00258 V=150.0 PL=0  +MOVJ EC00258
ARCON
SMOVL C00259 BC00259 V=9.2  +MOVJ EC00259
SMOVL C00260 BC00260 V=9.2  +MOVJ EC00260
SMOVL C00261 BC00261 V=9.2  +MOVJ EC00261
SMOVL C00262 BC00262 V=9.2  +MOVJ EC00262
SMOVL C00263 BC00263 V=9.2  +MOVJ EC00263
SMOVL C00264 BC00264 V=9.2  +MOVJ EC00264
ARCOF
SMOVL C00265 BC00265 V=800.0  +MOVJ EC00265
SMOVL C00266 BC00266 V=1000.0  +MOVJ EC00266
SFTOF3D
'EndPath W3636
'Path W4269
SFTOF3D
SFTON3D P024
MOVJ C00267 BC00267 VJ=100.00  +MOVJ EC00267 VJ=100.00
SMOVL C00268 BC00268 V=800.0  +MOVJ EC00268
SMOVL C00269 BC00269 V=150.0 PL=0  +MOVJ EC00269
ARCON
SMOVL C00270 BC00270 V=9.2  +MOVJ EC00270
SMOVL C00271 BC00271 V=9.2  +MOVJ EC00271
SMOVL C00272 BC00272 V=9.2  +MOVJ EC00272
SMOVL C00273 BC00273 V=9.2  +MOVJ EC00273
SMOVL C00274 BC00274 V=9.2  +MOVJ EC00274
SMOVL C00275 BC00275 V=9.2  +MOVJ EC00275
ARCOF
SMOVL C00276 BC00276 V=800.0  +MOVJ EC00276
SMOVL C00277 BC00277 V=1000.0  +MOVJ EC00277
SFTOF3D
MOVJ C00278 BC00278 VJ=100.00  +MOVJ EC00278 VJ=100.00
MOVJ C00279 BC00279 VJ=100.00  +MOVJ EC00279 VJ=100.00
SFTON3D P050
SMOVL C00280 BC00280 V=1000.0  +MOVJ EC00280
SMOVL C00281 BC00281 V=150.0 PL=0  +MOVJ EC00281
MACRO1 MJ#(0) ARGF9
ARCON
SMOVL C00282 BC00282 V=11.7  +MOVJ EC00282
SFTON3D P051
MOVL C00283 BC00283 V=11.7  +MOVJ EC00283 VJ=100.00
MOVL C00284 BC00284 V=11.7  +MOVJ EC00284 VJ=100.00
ARCOF
MOVL C00285 BC00285 V=166.7  +MOVJ EC00285 VJ=100.00
SFTOF3D
'EndPath W4269
MOVJ C00286 BC00286 VJ=100.00  +MOVJ EC00286 VJ=100.00
MOVJ C00287 BC00287 VJ=100.00  +MOVJ EC00287 VJ=100.00
MOVJ C00288 BC00288 VJ=100.00  +MOVJ EC00288 VJ=100.00
CALL JOB:CLEAN-R1_KM_3P
'
'
'
'Cut-Wire
MOVJ C00289 BC00289 VJ=100.00  +MOVJ EC00289 VJ=100.00
MOVJ C00290 BC00290 VJ=100.00  +MOVJ EC00290 VJ=100.00
MOVJ C00291 BC00291 VJ=100.00  +MOVJ EC00291 VJ=100.00
'obrot
MOVJ C00292 BC00292 VJ=100.00  +MOVJ EC00292 VJ=100.00
MOVJ C00293 BC00293 VJ=100.00  +MOVJ EC00293 VJ=100.00
MOVJ C00294 BC00294 VJ=100.00  +MOVJ EC00294 VJ=100.00
'Path S4271
SFTOF3D
MOVJ C00295 BC00295 VJ=100.00  +MOVJ EC00295 VJ=100.00
MOVL C00296 BC00296 V=800.0  +MOVJ EC00296 VJ=100.00
SMOVL C00297 BC00297 V=166.7  +MOVJ EC00297
SREFP 3 C00298 BC00298  +REFP EC00298
CALL JOB:SEARCH-R1-S13D
SET P021 P006
SFTON3D P021
SMOVL C00299 BC00299 V=166.7  +MOVJ EC00299
SREFP 3 C00300 BC00300  +REFP EC00300
CALL JOB:SEARCH-R1-S13D
SET P021 P006
SFTON3D P021
SMOVL C00301 BC00301 V=166.7  +MOVJ EC00301
'EndPath S4271
'Path S4272
SFTOF3D
MOVJ C00302 BC00302 VJ=100.00  +MOVJ EC00302 VJ=100.00
SMOVL C00303 BC00303 V=166.7  +MOVJ EC00303
SREFP 3 C00304 BC00304  +REFP EC00304
CALL JOB:SEARCH-R1-S13D
SET P022 P006
SFTON3D P022
SMOVL C00305 BC00305 V=166.7  +MOVJ EC00305
SMOVL C00306 BC00306 V=166.7  +MOVJ EC00306
SREFP 3 C00307 BC00307  +REFP EC00307
CALL JOB:SEARCH-R1-S13D
SET P022 P006
SFTON3D P022
SMOVL C00308 BC00308 V=166.7  +MOVJ EC00308
SMOVL C00309 BC00309 V=166.7  +MOVJ EC00309
SMOVL C00310 BC00310 V=166.7  +MOVJ EC00310
SREFP 3 C00311 BC00311  +REFP EC00311
CALL JOB:SEARCH-R1-S13D
SET P022 P006
SFTON3D P022
SMOVL C00312 BC00312 V=166.7  +MOVJ EC00312
'EndPath S4272
'Path S4273
SFTOF3D
MOVL C00313 BC00313 V=800.0  +MOVJ EC00313 VJ=100.00
SMOVL C00314 BC00314 V=166.7  +MOVJ EC00314
SREFP 3 C00315 BC00315  +REFP EC00315
CALL JOB:SEARCH-R1-S13D
SET P023 P006
SFTON3D P023
SMOVL C00316 BC00316 V=166.7  +MOVJ EC00316
SREFP 3 C00317 BC00317  +REFP EC00317
CALL JOB:SEARCH-R1-S13D
SET P023 P006
SFTON3D P023
SMOVL C00318 BC00318 V=166.7  +MOVJ EC00318
SMOVL C00319 BC00319 V=166.7  +MOVJ EC00319
SREFP 3 C00320 BC00320  +REFP EC00320
CALL JOB:SEARCH-R1-S13D
SET P023 P006
SFTON3D P023
SMOVL C00321 BC00321 V=166.7  +MOVJ EC00321
MOVL C00322 BC00322 V=1000.0  +MOVJ EC00322 VJ=100.00
'EndPath S4273
'Path S4274
SFTOF3D
MOVJ C00323 BC00323 VJ=100.00  +MOVJ EC00323 VJ=100.00
SMOVL C00324 BC00324 V=166.7  +MOVJ EC00324
SREFP 3 C00325 BC00325  +REFP EC00325
CALL JOB:SEARCH-R1-S13D
SET P024 P006
SFTON3D P024
SMOVL C00326 BC00326 V=166.7  +MOVJ EC00326
SREFP 3 C00327 BC00327  +REFP EC00327
CALL JOB:SEARCH-R1-S13D
SET P024 P006
SFTON3D P024
SMOVL C00328 BC00328 V=166.7  +MOVJ EC00328
SMOVL C00329 BC00329 V=166.7  +MOVJ EC00329
SMOVL C00330 BC00330 V=166.7  +MOVJ EC00330
SREFP 3 C00331 BC00331  +REFP EC00331
CALL JOB:SEARCH-R1-S13D
SET P024 P006
SFTON3D P024
SMOVL C00332 BC00332 V=166.7  +MOVJ EC00332
'EndPath S4274
'Path S4275
SFTOF3D
MOVL C00333 BC00333 V=800.0  +MOVJ EC00333 VJ=100.00
SMOVL C00334 BC00334 V=166.7  +MOVJ EC00334
SREFP 3 C00335 BC00335  +REFP EC00335
CALL JOB:SEARCH-R1-S13D
SET P025 P006
SFTON3D P025
SMOVL C00336 BC00336 V=166.7  +MOVJ EC00336
SMOVL C00337 BC00337 V=166.7  +MOVJ EC00337
SREFP 3 C00338 BC00338  +REFP EC00338
CALL JOB:SEARCH-R1-S13D
SET P025 P006
SFTON3D P025
SMOVL C00339 BC00339 V=166.7  +MOVJ EC00339
SMOVL C00340 BC00340 V=166.7  +MOVJ EC00340
SREFP 3 C00341 BC00341  +REFP EC00341
CALL JOB:SEARCH-R1-S13D
SET P025 P006
SFTON3D P025
SMOVL C00342 BC00342 V=166.7  +MOVJ EC00342
SFTOF3D
SMOVL C00343 BC00343 V=250.0  +MOVJ EC00343
SREFP 3 C00344 BC00344  +REFP EC00344
CALL JOB:SEARCH-R1-S13D
SET P026 P006
SFTON3D P026
SMOVL C00345 BC00345 V=166.7  +MOVJ EC00345
SREFP 3 C00346 BC00346  +REFP EC00346
CALL JOB:SEARCH-R1-S13D
SET P026 P006
SFTON3D P026
SMOVL C00347 BC00347 V=166.7  +MOVJ EC00347
SMOVL C00348 BC00348 V=250.0  +MOVJ EC00348
SMOVL C00349 BC00349 V=166.7  +MOVJ EC00349
SREFP 3 C00350 BC00350  +REFP EC00350
CALL JOB:SEARCH-R1-S13D
SET P026 P006
SFTON3D P026
SMOVL C00351 BC00351 V=166.7  +MOVJ EC00351
'EndPath S4276
'Path S4277
SFTOF3D
MOVL C00352 BC00352 V=800.0  +MOVJ EC00352 VJ=100.00
SMOVL C00353 BC00353 V=166.7  +MOVJ EC00353
SREFP 3 C00354 BC00354  +REFP EC00354
CALL JOB:SEARCH-R1-S13D
SET P027 P006
SFTON3D P027
SMOVL C00355 BC00355 V=166.7  +MOVJ EC00355
SMOVL C00356 BC00356 V=166.7  +MOVJ EC00356
SREFP 3 C00357 BC00357  +REFP EC00357
CALL JOB:SEARCH-R1-S13D
SET P027 P006
SFTON3D P027
SMOVL C00358 BC00358 V=166.7  +MOVJ EC00358
SMOVL C00359 BC00359 V=166.7  +MOVJ EC00359
SMOVL C00360 BC00360 V=166.7  +MOVJ EC00360
SREFP 3 C00361 BC00361  +REFP EC00361
CALL JOB:SEARCH-R1-S13D
SET P027 P006
SFTON3D P027
SMOVL C00362 BC00362 V=166.7  +MOVJ EC00362
SMOVL C00363 BC00363 V=166.7  +MOVJ EC00363
SMOVL C00364 BC00364 V=166.7  +MOVJ EC00364
MOVL C00365 BC00365 V=800.0  +MOVJ EC00365 VJ=100.00
MOVL C00366 BC00366 V=500.0  +MOVJ EC00366 VJ=100.00
SFTOF3D
MOVL C00367 BC00367 V=666.7  +MOVJ EC00367 VJ=0.78
SMOVL C00368 BC00368 V=166.7  +MOVJ EC00368
SREFP 3 C00369 BC00369  +REFP EC00369
CALL JOB:SEARCH-R1-S13D
SET P050 P006
SFTON3D P050
SMOVL C00370 BC00370 V=166.7  +MOVJ EC00370
SREFP 3 C00371 BC00371  +REFP EC00371
CALL JOB:SEARCH-R1-S13D
SET P050 P006
SFTON3D P050
SMOVL C00372 BC00372 V=166.7  +MOVJ EC00372
SFTOF3D
MOVL C00373 BC00373 V=666.7  +MOVJ EC00373 VJ=0.78
MOVL C00374 BC00374 V=666.7  +MOVJ EC00374 VJ=0.78
SMOVL C00375 BC00375 V=166.7  +MOVJ EC00375
SREFP 3 C00376 BC00376  +REFP EC00376
CALL JOB:SEARCH-R1-S13D
SET P051 P006
SFTON3D P051
SMOVL C00377 BC00377 V=166.7  +MOVJ EC00377
SREFP 3 C00378 BC00378  +REFP EC00378
CALL JOB:SEARCH-R1-S13D
SET P051 P006
SFTON3D P051
SMOVL C00379 BC00379 V=166.7  +MOVJ EC00379
SFTOF3D
MOVL C00380 BC00380 V=666.7  +MOVJ EC00380 VJ=0.78
MOVL C00381 BC00381 V=666.7  +MOVJ EC00381 VJ=0.78
MOVL C00382 BC00382 V=666.7  +MOVJ EC00382 VJ=0.78
MOVJ C00383 BC00383 VJ=100.00  +MOVJ EC00383 VJ=0.78
MOVL C00384 BC00384 V=666.7  +MOVJ EC00384 VJ=100.00
MOVL C00385 BC00385 V=666.7  +MOVJ EC00385 VJ=100.00
MOVL C00386 BC00386 V=666.7  +MOVJ EC00386 VJ=100.00
SFTON3D P051
SMOVL C00387 BC00387 V=166.7  +MOVJ EC00387
SREFP 3 C00388 BC00388  +REFP EC00388
CALL JOB:SEARCH-R1-S13D
SET P052 P006
SFTON3D P052
SMOVL C00389 BC00389 V=166.7  +MOVJ EC00389
SMOVL C00390 BC00390 V=166.7  +MOVJ EC00390
SMOVL C00391 BC00391 V=166.7  +MOVJ EC00391
SREFP 3 C00392 BC00392  +REFP EC00392
CALL JOB:SEARCH-R1-S13D
SET P052 P006
SFTON3D P052
SMOVL C00393 BC00393 V=166.7  +MOVJ EC00393
SMOVL C00394 BC00394 V=166.7  +MOVJ EC00394
SMOVL C00395 BC00395 V=166.7  +MOVJ EC00395
SREFP 3 C00396 BC00396  +REFP EC00396
CALL JOB:SEARCH-R1-S13D
SET P052 P006
SFTON3D P052
SMOVL C00397 BC00397 V=166.7  +MOVJ EC00397
SFTOF3D
MOVL C00398 BC00398 V=333.3  +MOVJ EC00398 VJ=100.00
SMOVL C00399 BC00399 V=166.7  +MOVJ EC00399
SREFP 3 C00400 BC00400  +REFP EC00400
CALL JOB:SEARCH-R1-S13D
SET P053 P006
SFTON3D P053
SMOVL C00401 BC00401 V=166.7  +MOVJ EC00401
SREFP 3 C00402 BC00402  +REFP EC00402
CALL JOB:SEARCH-R1-S13D
SET P053 P006
SFTON3D P053
SMOVL C00403 BC00403 V=166.7  +MOVJ EC00403
SFTOF3D
MOVL C00404 BC00404 V=333.3  +MOVJ EC00404 VJ=100.00
SFTON3D P052
SMOVL C00405 BC00405 V=166.7  +MOVJ EC00405
SREFP 3 C00406 BC00406  +REFP EC00406
CALL JOB:SEARCH-R1-S13D
SET P054 P006
SFTON3D P054
SMOVL C00407 BC00407 V=166.7  +MOVJ EC00407
SMOVL C00408 BC00408 V=166.7  +MOVJ EC00408
SMOVL C00409 BC00409 V=166.7  +MOVJ EC00409
SREFP 3 C00410 BC00410  +REFP EC00410
CALL JOB:SEARCH-R1-S13D
SET P054 P006
SFTON3D P054
SMOVL C00411 BC00411 V=166.7  +MOVJ EC00411
SMOVL C00412 BC00412 V=166.7  +MOVJ EC00412
SMOVL C00413 BC00413 V=166.7  +MOVJ EC00413
SREFP 3 C00414 BC00414  +REFP EC00414
CALL JOB:SEARCH-R1-S13D
SET P054 P006
SFTON3D P054
SMOVL C00415 BC00415 V=166.7  +MOVJ EC00415
SFTOF3D
MOVL C00416 BC00416 V=333.3  +MOVJ EC00416 VJ=100.00
MOVL C00417 BC00417 V=333.3  +MOVJ EC00417 VJ=100.00
SMOVL C00418 BC00418 V=166.7  +MOVJ EC00418
SREFP 3 C00419 BC00419  +REFP EC00419
CALL JOB:SEARCH-R1-S13D
SET P054 P006
SFTON3D P054
SMOVL C00420 BC00420 V=166.7  +MOVJ EC00420
SREFP 3 C00421 BC00421  +REFP EC00421
CALL JOB:SEARCH-R1-S13D
SET P054 P006
SFTON3D P054
SMOVL C00422 BC00422 V=166.7  +MOVJ EC00422
SFTOF3D
MOVL C00423 BC00423 V=333.3  +MOVJ EC00423 VJ=100.00
MOVL C00424 BC00424 V=333.3  +MOVJ EC00424 VJ=100.00
SFTON3D P052
MOVL C00425 BC00425 V=333.3  +MOVJ EC00425 VJ=100.00
MOVL C00426 BC00426 V=150.0 PL=0  +MOVJ EC00426 VJ=100.00
MACRO1 MJ#(0) ARGF9
ARCON
SMOVL C00427 BC00427 V=11.7  +MOVJ EC00427
SMOVC C00428 BC00428 V=13.3  +MOVJ EC00428
SMOVC C00429 BC00429 V=13.3  +MOVJ EC00429
SMOVC C00430 BC00430 V=13.3  +MOVJ EC00430
SMOVL C00431 BC00431 V=11.7  +MOVJ EC00431
SFTON3D P053
SMOVL C00432 BC00432 V=11.7  +MOVJ EC00432
ARCOF
SMOVL C00433 BC00433 V=166.7  +MOVJ EC00433
SFTOF3D
SMOVL C00434 BC00434 V=333.3  +MOVJ EC00434
MOVJ C00435 BC00435 VJ=30.00  +MOVJ EC00435 VJ=100.00
SFTON3D P054
SMOVL C00436 BC00436 V=333.3  +MOVJ EC00436
SMOVL C00437 BC00437 V=150.0 PL=0  +MOVJ EC00437
ARCON
SMOVL C00438 BC00438 V=11.7  +MOVJ EC00438
SMOVC C00439 BC00439 V=13.3  +MOVJ EC00439
SMOVC C00440 BC00440 V=13.3  +MOVJ EC00440
SMOVC C00441 BC00441 V=13.3  +MOVJ EC00441
SMOVL C00442 BC00442 V=11.7  +MOVJ EC00442
SFTON3D P055
SMOVL C00443 BC00443 V=11.7  +MOVJ EC00443
SMOVL C00444 BC00444 V=11.7  +MOVJ EC00444
ARCOF
SMOVL C00445 BC00445 V=166.7  +MOVJ EC00445
SFTOF3D
SMOVL C00446 BC00446 V=666.7  +MOVJ EC00446
MOVJ C00447 BC00447 VJ=30.00  +MOVJ EC00447 VJ=30.00
MOVJ C00448 BC00448 VJ=30.00  +MOVJ EC00448 VJ=30.00
MOVJ C00449 BC00449 VJ=30.00  +MOVJ EC00449 VJ=30.00
MOVJ C00450 BC00450 VJ=30.00  +MOVJ EC00450 VJ=30.00
MOVJ C00451 BC00451 VJ=30.00  +MOVJ EC00451 VJ=30.00
MOVJ C00452 BC00452 VJ=30.00  +MOVJ EC00452 VJ=30.00
'EndPath S4277
'
'Path W4278
SFTOF3D
SFTON3D P027
MOVJ C00453 BC00453 VJ=30.00  +MOVJ EC00453 VJ=30.00
MOVJ C00454 BC00454 VJ=30.00  +MOVJ EC00454 VJ=30.00
SMOVL C00455 BC00455 V=800.0  +MOVJ EC00455
SMOVL C00456 BC00456 V=150.0 PL=0  +MOVJ EC00456
ARCON
SMOVL C00457 BC00457 V=10.0  +MOVJ EC00457
SMOVL C00458 BC00458 V=10.0  +MOVJ EC00458
ARCOF
SMOVL C00459 BC00459 V=800.0  +MOVJ EC00459
SMOVL C00460 BC00460 V=1000.0  +MOVJ EC00460
SFTOF3D
'EndPath W4278
MOVJ C00461 BC00461 VJ=100.00  +MOVJ EC00461 VJ=100.00
MOVJ C00462 BC00462 VJ=100.00  +MOVJ EC00462 VJ=100.00
MOVJ C00463 BC00463 VJ=100.00  +MOVJ EC00463 VJ=100.00
'Path W4279
SFTOF3D
SFTON3D P021
MOVJ C00464 BC00464 VJ=100.00  +MOVJ EC00464 VJ=100.00
SMOVL C00465 BC00465 V=800.0  +MOVJ EC00465
SMOVL C00466 BC00466 V=150.0 PL=0  +MOVJ EC00466
SMOVL C00467 BC00467 V=10.0  +MOVJ EC00467
SMOVL C00468 BC00468 V=10.0  +MOVJ EC00468
SMOVL C00469 BC00469 V=10.0  +MOVJ EC00469
ARCOF
SMOVL C00470 BC00470 V=800.0  +MOVJ EC00470
SMOVL C00471 BC00471 V=1000.0  +MOVJ EC00471
SFTOF3D
'EndPath W4279
MOVJ C00472 BC00472 VJ=100.00  +MOVJ EC00472 VJ=100.00
SMOVL C00473 BC00473 V=500.0  +MOVJ EC00473
'Path W4280
SFTOF3D
SFTON3D P025
SMOVL C00474 BC00474 V=800.0  +MOVJ EC00474
SMOVL C00475 BC00475 V=150.0 PL=0  +MOVJ EC00475
ARCON
SMOVL C00476 BC00476 V=10.0  +MOVJ EC00476
SMOVL C00477 BC00477 V=10.0  +MOVJ EC00477
SMOVL C00478 BC00478 V=10.0  +MOVJ EC00478
SMOVL C00479 BC00479 V=10.0  +MOVJ EC00479
SMOVL C00480 BC00480 V=10.0  +MOVJ EC00480
SMOVL C00481 BC00481 V=10.0  +MOVJ EC00481
ARCOF
SMOVL C00482 BC00482 V=800.0  +MOVJ EC00482
SMOVL C00483 BC00483 V=1000.0  +MOVJ EC00483
SFTOF3D
'EndPath W4280
MOVJ C00484 BC00484 VJ=100.00  +MOVJ EC00484 VJ=100.00
'Path W4281
SFTOF3D
SFTON3D P023
MOVJ C00485 BC00485 VJ=100.00  +MOVJ EC00485 VJ=100.00
SMOVL C00486 BC00486 V=800.0  +MOVJ EC00486
SMOVL C00487 BC00487 V=150.0 PL=0  +MOVJ EC00487
ARCON
SMOVL C00488 BC00488 V=10.0  +MOVJ EC00488
SMOVL C00489 BC00489 V=10.0  +MOVJ EC00489
SMOVL C00490 BC00490 V=10.0  +MOVJ EC00490
SMOVL C00491 BC00491 V=10.0  +MOVJ EC00491
SMOVL C00492 BC00492 V=10.0  +MOVJ EC00492
SMOVL C00493 BC00493 V=10.0  +MOVJ EC00493
ARCOF
SMOVL C00494 BC00494 V=800.0  +MOVJ EC00494
SMOVL C00495 BC00495 V=1000.0  +MOVJ EC00495
SFTOF3D
'EndPath W4281
MOVJ C00496 BC00496 VJ=100.00  +MOVJ EC00496 VJ=100.00
'
'Path W4282
SFTOF3D
SFTON3D P026
MOVJ C00497 BC00497 VJ=100.00  +MOVJ EC00497 VJ=100.00
SMOVL C00498 BC00498 V=800.0  +MOVJ EC00498
SMOVL C00499 BC00499 V=150.0 PL=0  +MOVJ EC00499
ARCON
SMOVL C00500 BC00500 V=10.0  +MOVJ EC00500
SMOVL C00501 BC00501 V=10.0  +MOVJ EC00501
SMOVL C00502 BC00502 V=10.0  +MOVJ EC00502
SMOVL C00503 BC00503 V=10.0  +MOVJ EC00503
ARCOF
SMOVL C00504 BC00504 V=800.0  +MOVJ EC00504
SMOVL C00505 BC00505 V=1000.0  +MOVJ EC00505
SFTOF3D
'EndPath W4282
MOVJ C00506 BC00506 VJ=100.00  +MOVJ EC00506 VJ=100.00
MOVJ C00507 BC00507 VJ=100.00  +MOVJ EC00507 VJ=100.00
MOVJ C00508 BC00508 VJ=100.00  +MOVJ EC00508 VJ=100.00
'Path W4283
SFTOF3D
SFTON3D P022
MOVJ C00509 BC00509 VJ=100.00  +MOVJ EC00509 VJ=100.00
SMOVL C00510 BC00510 V=800.0  +MOVJ EC00510
SMOVL C00511 BC00511 V=150.0 PL=0  +MOVJ EC00511
ARCON
SMOVL C00512 BC00512 V=10.0  +MOVJ EC00512
SMOVL C00513 BC00513 V=10.0  +MOVJ EC00513
SMOVL C00514 BC00514 V=10.0  +MOVJ EC00514
SMOVL C00515 BC00515 V=10.0  +MOVJ EC00515
SMOVL C00516 BC00516 V=10.0  +MOVJ EC00516
SMOVL C00517 BC00517 V=10.0  +MOVJ EC00517
ARCOF
SMOVL C00518 BC00518 V=800.0  +MOVJ EC00518
SMOVL C00519 BC00519 V=1000.0  +MOVJ EC00519
SFTOF3D
'EndPath W4283
'Path W4284
SFTOF3D
SFTON3D P024
MOVJ C00520 BC00520 VJ=100.00  +MOVJ EC00520 VJ=100.00
SMOVL C00521 BC00521 V=800.0  +MOVJ EC00521
SMOVL C00522 BC00522 V=150.0 PL=0  +MOVJ EC00522
ARCON
SMOVL C00523 BC00523 V=10.0  +MOVJ EC00523
SMOVL C00524 BC00524 V=10.0  +MOVJ EC00524
SMOVL C00525 BC00525 V=10.0  +MOVJ EC00525
SMOVL C00526 BC00526 V=10.0  +MOVJ EC00526
SMOVL C00527 BC00527 V=10.0  +MOVJ EC00527
SMOVL C00528 BC00528 V=10.0  +MOVJ EC00528
ARCOF
SMOVL C00529 BC00529 V=800.0  +MOVJ EC00529
SMOVL C00530 BC00530 V=1000.0  +MOVJ EC00530
MOVJ C00531 BC00531 VJ=30.00  +MOVJ EC00531 VJ=30.00
MOVJ C00532 BC00532 VJ=30.00  +MOVJ EC00532 VJ=30.00
SFTON3D P051
SMOVL C00533 BC00533 V=150.0 PL=0  +MOVJ EC00533
MACRO1 MJ#(0) ARGF9
ARCON
SMOVL C00534 BC00534 V=11.7  +MOVJ EC00534
SFTON3D P050
SMOVL C00535 BC00535 V=11.7  +MOVJ EC00535
ARCOF
SMOVL C00536 BC00536 V=166.7  +MOVJ EC00536
SFTOF3D
'EndPath W4284
'
MOVJ C00537 BC00537 VJ=100.00  +MOVJ EC00537 VJ=100.00
MOVJ C00538 BC00538 VJ=100.00  +MOVJ EC00538 VJ=100.00
MOVJ C00539 BC00539 VJ=100.00  +MOVJ EC00539 VJ=100.00
'obrot
MOVJ C00540 BC00540 VJ=100.00  +MOVJ EC00540 VJ=100.00
MOVJ C00541 BC00541 VJ=100.00  +MOVJ EC00541 VJ=100.00
'
MOVJ C00542 BC00542 VJ=100.00  +MOVJ EC00542 VJ=100.00
'
END
